LIN {X 43.957,Y 37.252,Z 55.996,A 180.000,B 0.000,C 180.000} C_DIS
LIN {X 43.920,Y 37.565,Z 55.994,A 180.000,B 0.000,C 180.000} C_DIS
LIN {X 43.871,Y 37.876,Z 55.991,A 180.000,B 0.000,C 180.000} C_DIS
LIN {X 43.804,Y 38.184,Z 55.988,A 180.000,B 0.000,C 180.000} C_DIS
LIN {X 43.727,Y 38.489,Z 55.985,A 180.000,B 0.000,C 180.000} C_DIS
LIN {X 43.639,Y 38.792,Z 55.981,A 180.000,B 0.000,C 180.000} C_DIS
LIN {X 43.534,Y 39.089,Z 55.977,A 180.000,B 0.000,C 180.000} C_DIS
LIN {X 43.420,Y 39.382,Z 55.972,A 180.000,B 0.000,C 180.000} C_DIS
LIN {X 43.357,Y 39.527,Z 55.969,A 180.000,B 0.000,C 180.000} C_DIS
LIN {X 43.294,Y 39.671,Z 55.967,A 180.000,B 0.000,C 180.000} C_DIS
LIN {X 43.224,Y 39.812,Z 55.964,A 180.000,B 0.000,C 180.000} C_DIS
LIN {X 43.153,Y 39.952,Z 55.961,A 180.000,B 0.000,C 180.000} C_DIS
LIN {X 43.081,Y 40.093,Z 55.959,A 180.000,B 0.000,C 180.000} C_DIS
LIN {X 43.002,Y 40.229,Z 55.956,A 180.000,B 0.000,C 180.000} C_DIS
LIN {X 42.922,Y 40.365,Z 55.952,A 180.000,B 0.000,C 180.000} C_DIS
LIN {X 42.842,Y 40.500,Z 55.949,A 180.000,B 0.000,C 180.000} C_DIS
LIN {X 42.755,Y 40.631,Z 55.946,A 180.000,B 0.000,C 180.000} C_DIS
LIN {X 42.666,Y 40.761,Z 55.943,A 180.000,B 0.000,C 180.000} C_DIS
LIN {X 42.577,Y 40.892,Z 55.939,A 180.000,B 0.000,C 180.000} C_DIS
LIN {X 42.482,Y 41.017,Z 55.936,A 180.000,B 0.000,C 180.000} C_DIS
LIN {X 42.385,Y 41.141,Z 55.932,A 180.000,B 0.000,C 180.000} C_DIS
LIN {X 42.289,Y 41.266,Z 55.928,A 180.000,B 0.000,C 180.000} C_DIS
LIN {X 42.185,Y 41.385,Z 55.925,A 180.000,B 0.000,C 180.000} C_DIS
LIN {X 42.081,Y 41.503,Z 55.921,A 180.000,B 0.000,C 180.000} C_DIS
LIN {X 41.977,Y 41.621,Z 55.917,A 180.000,B 0.000,C 180.000} C_DIS
LIN {X 41.867,Y 41.733,Z 55.913,A 180.000,B 0.000,C 180.000} C_DIS
LIN {X 41.755,Y 41.844,Z 55.909,A 180.000,B 0.000,C 180.000} C_DIS
LIN {X 41.644,Y 41.956,Z 55.905,A 180.000,B 0.000,C 180.000} C_DIS
LIN {X 41.526,Y 42.061,Z 55.900,A 180.000,B 0.000,C 180.000} C_DIS
LIN {X 41.408,Y 42.165,Z 55.896,A 180.000,B 0.000,C 180.000} C_DIS
LIN {X 41.290,Y 42.269,Z 55.892,A 180.000,B 0.000,C 180.000} C_DIS
LIN {X 41.166,Y 42.366,Z 55.887,A 180.000,B 0.000,C 180.000} C_DIS
LIN {X 41.042,Y 42.463,Z 55.883,A 180.000,B 0.000,C 180.000} C_DIS
LIN {X 40.917,Y 42.559,Z 55.878,A 180.000,B 0.000,C 180.000} C_DIS
LIN {X 40.787,Y 42.648,Z 55.873,A 180.000,B 0.000,C 180.000} C_DIS
LIN {X 40.657,Y 42.737,Z 55.869,A 180.000,B 0.000,C 180.000} C_DIS
LIN {X 40.527,Y 42.826,Z 55.864,A 180.000,B 0.000,C 180.000} C_DIS
LIN {X 40.391,Y 42.906,Z 55.859,A 180.000,B 0.000,C 180.000} C_DIS
LIN {X 40.256,Y 42.986,Z 55.854,A 180.000,B 0.000,C 180.000} C_DIS
LIN {X 40.188,Y 43.027,Z 55.851,A 180.000,B 0.000,C 180.000} C_DIS
LIN {X 40.120,Y 43.067,Z 55.849,A 180.000,B 0.000,C 180.000} C_DIS
LIN {X 40.050,Y 43.103,Z 55.846,A 180.000,B 0.000,C 180.000} C_DIS
LIN {X 39.980,Y 43.139,Z 55.844,A 180.000,B 0.000,C 180.000} C_DIS
LIN {X 39.910,Y 43.174,Z 55.841,A 180.000,B 0.000,C 180.000} C_DIS
LIN {X 39.840,Y 43.210,Z 55.839,A 180.000,B 0.000,C 180.000} C_DIS
LIN {X 39.770,Y 43.246,Z 55.836,A 180.000,B 0.000,C 180.000} C_DIS
LIN {X 39.700,Y 43.282,Z 55.833,A 180.000,B 0.000,C 180.000} C_DIS
LIN {X 39.627,Y 43.313,Z 55.831,A 180.000,B 0.000,C 180.000} C_DIS
LIN {X 39.483,Y 43.376,Z 55.825,A 180.000,B 0.000,C 180.000} C_DIS
LIN {X 39.338,Y 43.438,Z 55.820,A 180.000,B 0.000,C 180.000} C_DIS
LIN {X 39.266,Y 43.470,Z 55.817,A 180.000,B 0.000,C 180.000} C_DIS
LIN {X 39.192,Y 43.497,Z 55.815,A 180.000,B 0.000,C 180.000} C_DIS
LIN {X 39.044,Y 43.550,Z 55.809,A 180.000,B 0.000,C 180.000} C_DIS
LIN {X 38.970,Y 43.577,Z 55.806,A 180.000,B 0.000,C 180.000} C_DIS
LIN {X 38.822,Y 43.630,Z 55.801,A 180.000,B 0.000,C 180.000} C_DIS
LIN {X 38.746,Y 43.652,Z 55.798,A 180.000,B 0.000,C 180.000} C_DIS
LIN {X 38.670,Y 43.674,Z 55.796,A 180.000,B 0.000,C 180.000} C_DIS
LIN {X 38.519,Y 43.718,Z 55.790,A 180.000,B 0.000,C 180.000} C_DIS
LIN {X 38.368,Y 43.762,Z 55.785,A 180.000,B 0.000,C 180.000} C_DIS
LIN {X 38.291,Y 43.780,Z 55.782,A 180.000,B 0.000,C 180.000} C_DIS
LIN {X 38.137,Y 43.814,Z 55.776,A 180.000,B 0.000,C 180.000} C_DIS
LIN {X 38.060,Y 43.831,Z 55.774,A 180.000,B 0.000,C 180.000} C_DIS
LIN {X 37.907,Y 43.866,Z 55.768,A 180.000,B 0.000,C 180.000} C_DIS
LIN {X 37.829,Y 43.878,Z 55.765,A 180.000,B 0.000,C 180.000} C_DIS
LIN {X 37.751,Y 43.890,Z 55.763,A 180.000,B 0.000,C 180.000} C_DIS
LIN {X 37.596,Y 43.915,Z 55.757,A 180.000,B 0.000,C 180.000} C_DIS
LIN {X 37.440,Y 43.940,Z 55.752,A 180.000,B 0.000,C 180.000} C_DIS
LIN {X 37.362,Y 43.947,Z 55.749,A 180.000,B 0.000,C 180.000} C_DIS
LIN {X 37.205,Y 43.962,Z 55.743,A 180.000,B 0.000,C 180.000} C_DIS
LIN {X 37.126,Y 43.969,Z 55.741,A 180.000,B 0.000,C 180.000} C_DIS
LIN {X 37.048,Y 43.977,Z 55.738,A 180.000,B 0.000,C 180.000} C_DIS
LIN {X 36.970,Y 43.984,Z 55.735,A 180.000,B 0.000,C 180.000} C_DIS
LIN {X 36.576,Y 43.996,Z 55.721,A 180.000,B 0.000,C 180.000} C_DIS
LIN {X 36.497,Y 43.999,Z 55.719,A 180.000,B 0.000,C 180.000} C_DIS
LIN {X 36.340,Y 43.994,Z 55.713,A 180.000,B 0.000,C 180.000} C_DIS
LIN {X 36.104,Y 43.986,Z 55.705,A 180.000,B 0.000,C 180.000} C_DIS
LIN {X 36.025,Y 43.984,Z 55.702,A 180.000,B 0.000,C 180.000} C_DIS
LIN {X 35.633,Y 43.947,Z 55.688,A 180.000,B 0.000,C 180.000} C_DIS
LIN {X 35.555,Y 43.939,Z 55.686,A 180.000,B 0.000,C 180.000} C_DIS
LIN {X 35.399,Y 43.914,Z 55.680,A 180.000,B 0.000,C 180.000} C_DIS
LIN {X 35.166,Y 43.877,Z 55.672,A 180.000,B 0.000,C 180.000} C_DIS
LIN {X 35.088,Y 43.864,Z 55.669,A 180.000,B 0.000,C 180.000} C_DIS
LIN {X 34.704,Y 43.778,Z 55.655,A 180.000,B 0.000,C 180.000} C_DIS
LIN {X 34.627,Y 43.761,Z 55.653,A 180.000,B 0.000,C 180.000} C_DIS
LIN {X 34.400,Y 43.695,Z 55.644,A 180.000,B 0.000,C 180.000} C_DIS
LIN {X 34.249,Y 43.651,Z 55.639,A 180.000,B 0.000,C 180.000} C_DIS
LIN {X 34.173,Y 43.628,Z 55.636,A 180.000,B 0.000,C 180.000} C_DIS
LIN {X 33.803,Y 43.495,Z 55.622,A 180.000,B 0.000,C 180.000} C_DIS
LIN {X 33.729,Y 43.468,Z 55.620,A 180.000,B 0.000,C 180.000} C_DIS
LIN {X 33.512,Y 43.374,Z 55.611,A 180.000,B 0.000,C 180.000} C_DIS
LIN {X 33.368,Y 43.311,Z 55.606,A 180.000,B 0.000,C 180.000} C_DIS
LIN {X 33.296,Y 43.279,Z 55.603,A 180.000,B 0.000,C 180.000} C_DIS
LIN {X 32.945,Y 43.100,Z 55.589,A 180.000,B 0.000,C 180.000} C_DIS
LIN {X 32.875,Y 43.064,Z 55.587,A 180.000,B 0.000,C 180.000} C_DIS
LIN {X 32.536,Y 42.863,Z 55.573,A 180.000,B 0.000,C 180.000} C_DIS
LIN {X 32.469,Y 42.822,Z 55.570,A 180.000,B 0.000,C 180.000} C_DIS
LIN {X 32.143,Y 42.601,Z 55.556,A 180.000,B 0.000,C 180.000} C_DIS
LIN {X 32.079,Y 42.556,Z 55.554,A 180.000,B 0.000,C 180.000} C_DIS
LIN {X 31.767,Y 42.315,Z 55.540,A 180.000,B 0.000,C 180.000} C_DIS
LIN {X 31.706,Y 42.265,Z 55.537,A 180.000,B 0.000,C 180.000} C_DIS
LIN {X 31.410,Y 42.005,Z 55.523,A 180.000,B 0.000,C 180.000} C_DIS
LIN {X 31.352,Y 41.952,Z 55.521,A 180.000,B 0.000,C 180.000} C_DIS
LIN {X 31.074,Y 41.673,Z 55.507,A 180.000,B 0.000,C 180.000} C_DIS
LIN {X 31.019,Y 41.617,Z 55.504,A 180.000,B 0.000,C 180.000} C_DIS
LIN {X 30.759,Y 41.321,Z 55.490,A 180.000,B 0.000,C 180.000} C_DIS
LIN {X 30.708,Y 41.261,Z 55.488,A 180.000,B 0.000,C 180.000} C_DIS
LIN {X 30.466,Y 40.950,Z 55.474,A 180.000,B 0.000,C 180.000} C_DIS
LIN {X 30.419,Y 40.887,Z 55.471,A 180.000,B 0.000,C 180.000} C_DIS
LIN {X 30.198,Y 40.561,Z 55.457,A 180.000,B 0.000,C 180.000} C_DIS
LIN {X 30.155,Y 40.495,Z 55.455,A 180.000,B 0.000,C 180.000} C_DIS
LIN {X 29.955,Y 40.156,Z 55.441,A 180.000,B 0.000,C 180.000} C_DIS
LIN {X 29.916,Y 40.088,Z 55.438,A 180.000,B 0.000,C 180.000} C_DIS
LIN {X 29.737,Y 39.737,Z 55.424,A 180.000,B 0.000,C 180.000} C_DIS
LIN {X 29.703,Y 39.666,Z 55.422,A 180.000,B 0.000,C 180.000} C_DIS
LIN {X 29.547,Y 39.305,Z 55.408,A 180.000,B 0.000,C 180.000} C_DIS
LIN {X 29.517,Y 39.232,Z 55.405,A 180.000,B 0.000,C 180.000} C_DIS
LIN {X 29.384,Y 38.861,Z 55.391,A 180.000,B 0.000,C 180.000} C_DIS
LIN {X 29.359,Y 38.786,Z 55.389,A 180.000,B 0.000,C 180.000} C_DIS
LIN {X 29.293,Y 38.559,Z 55.380,A 180.000,B 0.000,C 180.000} C_DIS
LIN {X 29.249,Y 38.408,Z 55.375,A 180.000,B 0.000,C 180.000} C_DIS
LIN {X 29.229,Y 38.332,Z 55.372,A 180.000,B 0.000,C 180.000} C_DIS
LIN {X 29.144,Y 37.948,Z 55.358,A 180.000,B 0.000,C 180.000} C_DIS
LIN {X 29.129,Y 37.870,Z 55.356,A 180.000,B 0.000,C 180.000} C_DIS
LIN {X 29.092,Y 37.637,Z 55.347,A 180.000,B 0.000,C 180.000} C_DIS
LIN {X 29.067,Y 37.481,Z 55.342,A 180.000,B 0.000,C 180.000} C_DIS
LIN {X 29.057,Y 37.403,Z 55.339,A 180.000,B 0.000,C 180.000} C_DIS
LIN {X 29.020,Y 37.011,Z 55.325,A 180.000,B 0.000,C 180.000} C_DIS
LIN {X 29.015,Y 36.933,Z 55.323,A 180.000,B 0.000,C 180.000} C_DIS
LIN {X 29.010,Y 36.775,Z 55.317,A 180.000,B 0.000,C 180.000} C_DIS
LIN {X 29.002,Y 36.539,Z 55.309,A 180.000,B 0.000,C 180.000} C_DIS
LIN {X 29.002,Y 36.460,Z 55.306,A 180.000,B 0.000,C 180.000} C_DIS
LIN {X 29.015,Y 36.067,Z 55.292,A 180.000,B 0.000,C 180.000} C_DIS
LIN {X 29.020,Y 35.988,Z 55.290,A 180.000,B 0.000,C 180.000} C_DIS
LIN {X 29.035,Y 35.831,Z 55.284,A 180.000,B 0.000,C 180.000} C_DIS
LIN {X 29.057,Y 35.596,Z 55.276,A 180.000,B 0.000,C 180.000} C_DIS
LIN {X 29.067,Y 35.518,Z 55.273,A 180.000,B 0.000,C 180.000} C_DIS
LIN {X 29.104,Y 35.285,Z 55.265,A 180.000,B 0.000,C 180.000} C_DIS
LIN {X 29.129,Y 35.129,Z 55.259,A 180.000,B 0.000,C 180.000} C_DIS
LIN {X 29.144,Y 35.052,Z 55.257,A 180.000,B 0.000,C 180.000} C_DIS
LIN {X 29.178,Y 34.898,Z 55.251,A 180.000,B 0.000,C 180.000} C_DIS
LIN {X 29.230,Y 34.668,Z 55.243,A 180.000,B 0.000,C 180.000} C_DIS
LIN {X 29.250,Y 34.591,Z 55.240,A 180.000,B 0.000,C 180.000} C_DIS
LIN {X 29.315,Y 34.365,Z 55.232,A 180.000,B 0.000,C 180.000} C_DIS
LIN {X 29.359,Y 34.213,Z 55.226,A 180.000,B 0.000,C 180.000} C_DIS
LIN {X 29.384,Y 34.139,Z 55.224,A 180.000,B 0.000,C 180.000} C_DIS
LIN {X 29.438,Y 33.990,Z 55.218,A 180.000,B 0.000,C 180.000} C_DIS
LIN {X 29.518,Y 33.768,Z 55.210,A 180.000,B 0.000,C 180.000} C_DIS
LIN {X 29.547,Y 33.695,Z 55.207,A 180.000,B 0.000,C 180.000} C_DIS
LIN {X 29.641,Y 33.478,Z 55.199,A 180.000,B 0.000,C 180.000} C_DIS
LIN {X 29.703,Y 33.334,Z 55.193,A 180.000,B 0.000,C 180.000} C_DIS
LIN {X 29.738,Y 33.263,Z 55.191,A 180.000,B 0.000,C 180.000} C_DIS
LIN {X 29.809,Y 33.122,Z 55.185,A 180.000,B 0.000,C 180.000} C_DIS
LIN {X 29.881,Y 32.982,Z 55.180,A 180.000,B 0.000,C 180.000} C_DIS
LIN {X 29.916,Y 32.912,Z 55.177,A 180.000,B 0.000,C 180.000} C_DIS
LIN {X 29.955,Y 32.843,Z 55.174,A 180.000,B 0.000,C 180.000} C_DIS
LIN {X 30.035,Y 32.708,Z 55.169,A 180.000,B 0.000,C 180.000} C_DIS
LIN {X 30.115,Y 32.572,Z 55.164,A 180.000,B 0.000,C 180.000} C_DIS
LIN {X 30.155,Y 32.504,Z 55.161,A 180.000,B 0.000,C 180.000} C_DIS
LIN {X 30.198,Y 32.438,Z 55.159,A 180.000,B 0.000,C 180.000} C_DIS
LIN {X 30.243,Y 32.373,Z 55.156,A 180.000,B 0.000,C 180.000} C_DIS
LIN {X 30.287,Y 32.308,Z 55.154,A 180.000,B 0.000,C 180.000} C_DIS
LIN {X 30.331,Y 32.243,Z 55.151,A 180.000,B 0.000,C 180.000} C_DIS
LIN {X 30.375,Y 32.178,Z 55.149,A 180.000,B 0.000,C 180.000} C_DIS
LIN {X 30.467,Y 32.049,Z 55.144,A 180.000,B 0.000,C 180.000} C_DIS
LIN {X 30.563,Y 31.925,Z 55.139,A 180.000,B 0.000,C 180.000} C_DIS
LIN {X 30.660,Y 31.800,Z 55.134,A 180.000,B 0.000,C 180.000} C_DIS
LIN {X 30.759,Y 31.678,Z 55.129,A 180.000,B 0.000,C 180.000} C_DIS
LIN {X 30.863,Y 31.560,Z 55.124,A 180.000,B 0.000,C 180.000} C_DIS
LIN {X 30.967,Y 31.442,Z 55.120,A 180.000,B 0.000,C 180.000} C_DIS
LIN {X 31.074,Y 31.326,Z 55.115,A 180.000,B 0.000,C 180.000} C_DIS
LIN {X 31.186,Y 31.215,Z 55.111,A 180.000,B 0.000,C 180.000} C_DIS
LIN {X 31.297,Y 31.103,Z 55.106,A 180.000,B 0.000,C 180.000} C_DIS
LIN {X 31.411,Y 30.995,Z 55.102,A 180.000,B 0.000,C 180.000} C_DIS
LIN {X 31.529,Y 30.891,Z 55.097,A 180.000,B 0.000,C 180.000} C_DIS
LIN {X 31.647,Y 30.786,Z 55.093,A 180.000,B 0.000,C 180.000} C_DIS
LIN {X 31.768,Y 30.685,Z 55.089,A 180.000,B 0.000,C 180.000} C_DIS
LIN {X 31.892,Y 30.589,Z 55.085,A 180.000,B 0.000,C 180.000} C_DIS
LIN {X 32.017,Y 30.492,Z 55.081,A 180.000,B 0.000,C 180.000} C_DIS
LIN {X 32.144,Y 30.399,Z 55.077,A 180.000,B 0.000,C 180.000} C_DIS
LIN {X 32.274,Y 30.310,Z 55.073,A 180.000,B 0.000,C 180.000} C_DIS
LIN {X 32.404,Y 30.222,Z 55.070,A 180.000,B 0.000,C 180.000} C_DIS
LIN {X 32.537,Y 30.136,Z 55.066,A 180.000,B 0.000,C 180.000} C_DIS
LIN {X 32.672,Y 30.056,Z 55.062,A 180.000,B 0.000,C 180.000} C_DIS
LIN {X 32.808,Y 29.976,Z 55.059,A 180.000,B 0.000,C 180.000} C_DIS
LIN {X 32.945,Y 29.899,Z 55.056,A 180.000,B 0.000,C 180.000} C_DIS
LIN {X 33.086,Y 29.828,Z 55.052,A 180.000,B 0.000,C 180.000} C_DIS
LIN {X 33.226,Y 29.756,Z 55.049,A 180.000,B 0.000,C 180.000} C_DIS
LIN {X 33.368,Y 29.689,Z 55.046,A 180.000,B 0.000,C 180.000} C_DIS
LIN {X 33.513,Y 29.626,Z 55.043,A 180.000,B 0.000,C 180.000} C_DIS
LIN {X 33.657,Y 29.563,Z 55.040,A 180.000,B 0.000,C 180.000} C_DIS
LIN {X 33.803,Y 29.505,Z 55.037,A 180.000,B 0.000,C 180.000} C_DIS
LIN {X 33.952,Y 29.451,Z 55.034,A 180.000,B 0.000,C 180.000} C_DIS
LIN {X 34.100,Y 29.398,Z 55.032,A 180.000,B 0.000,C 180.000} C_DIS
LIN {X 34.249,Y 29.349,Z 55.029,A 180.000,B 0.000,C 180.000} C_DIS
LIN {X 34.401,Y 29.305,Z 55.027,A 180.000,B 0.000,C 180.000} C_DIS
LIN {X 34.704,Y 29.221,Z 55.022,A 180.000,B 0.000,C 180.000} C_DIS
LIN {X 35.012,Y 29.153,Z 55.018,A 180.000,B 0.000,C 180.000} C_DIS
LIN {X 35.322,Y 29.098,Z 55.014,A 180.000,B 0.000,C 180.000} C_DIS
LIN {X 35.634,Y 29.053,Z 55.011,A 180.000,B 0.000,C 180.000} C_DIS
LIN {X 35.947,Y 29.024,Z 55.008,A 180.000,B 0.000,C 180.000} C_DIS
LIN {X 36.262,Y 29.009,Z 55.005,A 180.000,B 0.000,C 180.000} C_DIS
LIN {X 36.577,Y 29.004,Z 55.003,A 180.000,B 0.000,C 180.000} C_DIS
LIN {X 36.891,Y 29.014,Z 55.002,A 180.000,B 0.000,C 180.000} C_DIS
LIN {X 37.205,Y 29.038,Z 55.001,A 180.000,B 0.000,C 180.000} C_DIS
LIN {X 37.518,Y 29.073,Z 55.000,A 180.000,B 0.000,C 180.000} C_DIS
LIN {X 37.748,Y 29.109,Z 55.000,A 180.000,B 0.000,C 180.000} C_DIS
; Cutting Move Starts
LIN {X 37.902,Y 29.134,Z 55.000,A 180.000,B 0.000,C 180.000} C_DIS
LIN {X 37.944,Y 29.143,Z 55.000,A 180.000,B 0.000,C 180.000} C_DIS
LIN {X 38.260,Y 29.213,Z 55.000,A 180.000,B 0.000,C 180.000} C_DIS
LIN {X 38.439,Y 29.258,Z 55.000,A 180.000,B 0.000,C 180.000} C_DIS
LIN {X 38.796,Y 29.362,Z 55.000,A 180.000,B 0.000,C 180.000} C_DIS
LIN {X 38.975,Y 29.425,Z 55.000,A 180.000,B 0.000,C 180.000} C_DIS
LIN {X 39.184,Y 29.500,Z 55.000,A 180.000,B 0.000,C 180.000} C_DIS
LIN {X 39.333,Y 29.559,Z 55.000,A 180.000,B 0.000,C 180.000} C_DIS
LIN {X 39.690,Y 29.714,Z 55.000,A 180.000,B 0.000,C 180.000} C_DIS
LIN {X 39.869,Y 29.805,Z 55.000,A 180.000,B 0.000,C 180.000} C_DIS
LIN {X 40.048,Y 29.896,Z 55.000,A 180.000,B 0.000,C 180.000} C_DIS
LIN {X 40.226,Y 29.996,Z 55.000,A 180.000,B 0.000,C 180.000} C_DIS
LIN {X 40.405,Y 30.102,Z 55.000,A 180.000,B 0.000,C 180.000} C_DIS
LIN {X 40.584,Y 30.213,Z 55.000,A 180.000,B 0.000,C 180.000} C_DIS
LIN {X 40.850,Y 30.394,Z 55.000,A 180.000,B 0.000,C 180.000} C_DIS
LIN {X 40.942,Y 30.460,Z 55.000,A 180.000,B 0.000,C 180.000} C_DIS
LIN {X 41.120,Y 30.598,Z 55.000,A 180.000,B 0.000,C 180.000} C_DIS
LIN {X 41.299,Y 30.739,Z 55.000,A 180.000,B 0.000,C 180.000} C_DIS
LIN {X 41.516,Y 30.930,Z 55.000,A 180.000,B 0.000,C 180.000} C_DIS
LIN {X 41.657,Y 31.057,Z 55.000,A 180.000,B 0.000,C 180.000} C_DIS
LIN {X 41.888,Y 31.288,Z 55.000,A 180.000,B 0.000,C 180.000} C_DIS
LIN {X 42.014,Y 31.421,Z 55.000,A 180.000,B 0.000,C 180.000} C_DIS
LIN {X 42.212,Y 31.646,Z 55.000,A 180.000,B 0.000,C 180.000} C_DIS
LIN {X 42.359,Y 31.824,Z 55.000,A 180.000,B 0.000,C 180.000} C_DIS
LIN {X 42.550,Y 32.072,Z 55.000,A 180.000,B 0.000,C 180.000} C_DIS
LIN {X 42.627,Y 32.182,Z 55.000,A 180.000,B 0.000,C 180.000} C_DIS
LIN {X 42.749,Y 32.361,Z 55.000,A 180.000,B 0.000,C 180.000} C_DIS
LIN {X 42.865,Y 32.539,Z 55.000,A 180.000,B 0.000,C 180.000} C_DIS
LIN {X 42.971,Y 32.718,Z 55.000,A 180.000,B 0.000,C 180.000} C_DIS
LIN {X 43.076,Y 32.897,Z 55.000,A 180.000,B 0.000,C 180.000} C_DIS
LIN {X 43.266,Y 33.269,Z 55.000,A 180.000,B 0.000,C 180.000} C_DIS
LIN {X 43.340,Y 33.433,Z 55.000,A 180.000,B 0.000,C 180.000} C_DIS
LIN {X 43.444,Y 33.675,Z 55.000,A 180.000,B 0.000,C 180.000} C_DIS
LIN {X 43.491,Y 33.791,Z 55.000,A 180.000,B 0.000,C 180.000} C_DIS
LIN {X 43.623,Y 34.159,Z 55.000,A 180.000,B 0.000,C 180.000} C_DIS
LIN {X 43.674,Y 34.327,Z 55.000,A 180.000,B 0.000,C 180.000} C_DIS
LIN {X 43.726,Y 34.506,Z 55.000,A 180.000,B 0.000,C 180.000} C_DIS
LIN {X 43.774,Y 34.685,Z 55.000,A 180.000,B 0.000,C 180.000} C_DIS
LIN {X 43.854,Y 35.042,Z 55.000,A 180.000,B 0.000,C 180.000} C_DIS
LIN {X 43.886,Y 35.221,Z 55.000,A 180.000,B 0.000,C 180.000} C_DIS
LIN {X 43.914,Y 35.400,Z 55.000,A 180.000,B 0.000,C 180.000} C_DIS
LIN {X 43.941,Y 35.578,Z 55.000,A 180.000,B 0.000,C 180.000} C_DIS
LIN {X 43.981,Y 35.994,Z 55.000,A 180.000,B 0.000,C 180.000} C_DIS
LIN {X 43.987,Y 36.115,Z 55.000,A 180.000,B 0.000,C 180.000} C_DIS
LIN {X 43.998,Y 36.472,Z 55.000,A 180.000,B 0.000,C 180.000} C_DIS
LIN {X 43.994,Y 36.651,Z 55.000,A 180.000,B 0.000,C 180.000} C_DIS
LIN {X 43.988,Y 36.830,Z 55.000,A 180.000,B 0.000,C 180.000} C_DIS
LIN {X 43.981,Y 37.006,Z 55.000,A 180.000,B 0.000,C 180.000} C_DIS
LIN {X 43.947,Y 37.366,Z 55.000,A 180.000,B 0.000,C 180.000} C_DIS
LIN {X 43.923,Y 37.545,Z 55.000,A 180.000,B 0.000,C 180.000} C_DIS
LIN {X 43.866,Y 37.902,Z 55.000,A 180.000,B 0.000,C 180.000} C_DIS
LIN {X 43.827,Y 38.081,Z 55.000,A 180.000,B 0.000,C 180.000} C_DIS
LIN {X 43.787,Y 38.260,Z 55.000,A 180.000,B 0.000,C 180.000} C_DIS
LIN {X 43.742,Y 38.439,Z 55.000,A 180.000,B 0.000,C 180.000} C_DIS
LIN {X 43.638,Y 38.796,Z 55.000,A 180.000,B 0.000,C 180.000} C_DIS
LIN {X 43.623,Y 38.841,Z 55.000,A 180.000,B 0.000,C 180.000} C_DIS
LIN {X 43.511,Y 39.154,Z 55.000,A 180.000,B 0.000,C 180.000} C_DIS
LIN {X 43.444,Y 39.325,Z 55.000,A 180.000,B 0.000,C 180.000} C_DIS
LIN {X 43.286,Y 39.690,Z 55.000,A 180.000,B 0.000,C 180.000} C_DIS
LIN {X 43.266,Y 39.731,Z 55.000,A 180.000,B 0.000,C 180.000} C_DIS
LIN {X 43.087,Y 40.082,Z 55.000,A 180.000,B 0.000,C 180.000} C_DIS
LIN {X 43.004,Y 40.226,Z 55.000,A 180.000,B 0.000,C 180.000} C_DIS
LIN {X 42.898,Y 40.405,Z 55.000,A 180.000,B 0.000,C 180.000} C_DIS
LIN {X 42.787,Y 40.584,Z 55.000,A 180.000,B 0.000,C 180.000} C_DIS
LIN {X 42.665,Y 40.763,Z 55.000,A 180.000,B 0.000,C 180.000} C_DIS
LIN {X 42.550,Y 40.928,Z 55.000,A 180.000,B 0.000,C 180.000} C_DIS
LIN {X 42.372,Y 41.159,Z 55.000,A 180.000,B 0.000,C 180.000} C_DIS
LIN {X 42.261,Y 41.299,Z 55.000,A 180.000,B 0.000,C 180.000} C_DIS
LIN {X 42.014,Y 41.579,Z 55.000,A 180.000,B 0.000,C 180.000} C_DIS
LIN {X 41.943,Y 41.657,Z 55.000,A 180.000,B 0.000,C 180.000} C_DIS
LIN {X 41.657,Y 41.943,Z 55.000,A 180.000,B 0.000,C 180.000} C_DIS
LIN {X 41.579,Y 42.014,Z 55.000,A 180.000,B 0.000,C 180.000} C_DIS
LIN {X 41.299,Y 42.261,Z 55.000,A 180.000,B 0.000,C 180.000} C_DIS
LIN {X 41.159,Y 42.372,Z 55.000,A 180.000,B 0.000,C 180.000} C_DIS
LIN {X 40.928,Y 42.550,Z 55.000,A 180.000,B 0.000,C 180.000} C_DIS
LIN {X 40.763,Y 42.665,Z 55.000,A 180.000,B 0.000,C 180.000} C_DIS
LIN {X 40.584,Y 42.787,Z 55.000,A 180.000,B 0.000,C 180.000} C_DIS
LIN {X 40.405,Y 42.898,Z 55.000,A 180.000,B 0.000,C 180.000} C_DIS
LIN {X 40.226,Y 43.004,Z 55.000,A 180.000,B 0.000,C 180.000} C_DIS
LIN {X 40.082,Y 43.087,Z 55.000,A 180.000,B 0.000,C 180.000} C_DIS
LIN {X 39.731,Y 43.266,Z 55.000,A 180.000,B 0.000,C 180.000} C_DIS
LIN {X 39.690,Y 43.286,Z 55.000,A 180.000,B 0.000,C 180.000} C_DIS
LIN {X 39.325,Y 43.444,Z 55.000,A 180.000,B 0.000,C 180.000} C_DIS
LIN {X 39.154,Y 43.511,Z 55.000,A 180.000,B 0.000,C 180.000} C_DIS
LIN {X 38.841,Y 43.623,Z 55.000,A 180.000,B 0.000,C 180.000} C_DIS
LIN {X 38.796,Y 43.638,Z 55.000,A 180.000,B 0.000,C 180.000} C_DIS
LIN {X 38.439,Y 43.742,Z 55.000,A 180.000,B 0.000,C 180.000} C_DIS
LIN {X 38.260,Y 43.787,Z 55.000,A 180.000,B 0.000,C 180.000} C_DIS
LIN {X 38.081,Y 43.827,Z 55.000,A 180.000,B 0.000,C 180.000} C_DIS
LIN {X 37.902,Y 43.866,Z 55.000,A 180.000,B 0.000,C 180.000} C_DIS
LIN {X 37.545,Y 43.923,Z 55.000,A 180.000,B 0.000,C 180.000} C_DIS
LIN {X 37.366,Y 43.947,Z 55.000,A 180.000,B 0.000,C 180.000} C_DIS
LIN {X 37.006,Y 43.981,Z 55.000,A 180.000,B 0.000,C 180.000} C_DIS
LIN {X 36.830,Y 43.988,Z 55.000,A 180.000,B 0.000,C 180.000} C_DIS
LIN {X 36.651,Y 43.994,Z 55.000,A 180.000,B 0.000,C 180.000} C_DIS
LIN {X 36.472,Y 43.998,Z 55.000,A 180.000,B 0.000,C 180.000} C_DIS
LIN {X 36.115,Y 43.987,Z 55.000,A 180.000,B 0.000,C 180.000} C_DIS
LIN {X 35.994,Y 43.981,Z 55.000,A 180.000,B 0.000,C 180.000} C_DIS
LIN {X 35.578,Y 43.941,Z 55.000,A 180.000,B 0.000,C 180.000} C_DIS
LIN {X 35.400,Y 43.914,Z 55.000,A 180.000,B 0.000,C 180.000} C_DIS
LIN {X 35.221,Y 43.886,Z 55.000,A 180.000,B 0.000,C 180.000} C_DIS
LIN {X 35.042,Y 43.854,Z 55.000,A 180.000,B 0.000,C 180.000} C_DIS
LIN {X 34.685,Y 43.774,Z 55.000,A 180.000,B 0.000,C 180.000} C_DIS
LIN {X 34.506,Y 43.726,Z 55.000,A 180.000,B 0.000,C 180.000} C_DIS
LIN {X 34.327,Y 43.674,Z 55.000,A 180.000,B 0.000,C 180.000} C_DIS
LIN {X 34.159,Y 43.623,Z 55.000,A 180.000,B 0.000,C 180.000} C_DIS
LIN {X 33.791,Y 43.491,Z 55.000,A 180.000,B 0.000,C 180.000} C_DIS
LIN {X 33.675,Y 43.444,Z 55.000,A 180.000,B 0.000,C 180.000} C_DIS
LIN {X 33.433,Y 43.340,Z 55.000,A 180.000,B 0.000,C 180.000} C_DIS
LIN {X 33.269,Y 43.266,Z 55.000,A 180.000,B 0.000,C 180.000} C_DIS
LIN {X 32.897,Y 43.076,Z 55.000,A 180.000,B 0.000,C 180.000} C_DIS
LIN {X 32.718,Y 42.971,Z 55.000,A 180.000,B 0.000,C 180.000} C_DIS
LIN {X 32.539,Y 42.865,Z 55.000,A 180.000,B 0.000,C 180.000} C_DIS
LIN {X 32.361,Y 42.749,Z 55.000,A 180.000,B 0.000,C 180.000} C_DIS
LIN {X 32.182,Y 42.627,Z 55.000,A 180.000,B 0.000,C 180.000} C_DIS
LIN {X 32.072,Y 42.550,Z 55.000,A 180.000,B 0.000,C 180.000} C_DIS
LIN {X 31.824,Y 42.359,Z 55.000,A 180.000,B 0.000,C 180.000} C_DIS
LIN {X 31.646,Y 42.212,Z 55.000,A 180.000,B 0.000,C 180.000} C_DIS
LIN {X 31.421,Y 42.014,Z 55.000,A 180.000,B 0.000,C 180.000} C_DIS
LIN {X 31.288,Y 41.888,Z 55.000,A 180.000,B 0.000,C 180.000} C_DIS
LIN {X 31.057,Y 41.657,Z 55.000,A 180.000,B 0.000,C 180.000} C_DIS
LIN {X 30.930,Y 41.516,Z 55.000,A 180.000,B 0.000,C 180.000} C_DIS
LIN {X 30.739,Y 41.299,Z 55.000,A 180.000,B 0.000,C 180.000} C_DIS
LIN {X 30.598,Y 41.120,Z 55.000,A 180.000,B 0.000,C 180.000} C_DIS
LIN {X 30.460,Y 40.942,Z 55.000,A 180.000,B 0.000,C 180.000} C_DIS
LIN {X 30.394,Y 40.850,Z 55.000,A 180.000,B 0.000,C 180.000} C_DIS
LIN {X 30.213,Y 40.584,Z 55.000,A 180.000,B 0.000,C 180.000} C_DIS
LIN {X 30.102,Y 40.405,Z 55.000,A 180.000,B 0.000,C 180.000} C_DIS
LIN {X 29.996,Y 40.226,Z 55.000,A 180.000,B 0.000,C 180.000} C_DIS
LIN {X 29.896,Y 40.048,Z 55.000,A 180.000,B 0.000,C 180.000} C_DIS
LIN {X 29.805,Y 39.869,Z 55.000,A 180.000,B 0.000,C 180.000} C_DIS
LIN {X 29.714,Y 39.690,Z 55.000,A 180.000,B 0.000,C 180.000} C_DIS
LIN {X 29.559,Y 39.333,Z 55.000,A 180.000,B 0.000,C 180.000} C_DIS
LIN {X 29.500,Y 39.184,Z 55.000,A 180.000,B 0.000,C 180.000} C_DIS
LIN {X 29.425,Y 38.975,Z 55.000,A 180.000,B 0.000,C 180.000} C_DIS
LIN {X 29.362,Y 38.796,Z 55.000,A 180.000,B 0.000,C 180.000} C_DIS
LIN {X 29.258,Y 38.439,Z 55.000,A 180.000,B 0.000,C 180.000} C_DIS
LIN {X 29.213,Y 38.260,Z 55.000,A 180.000,B 0.000,C 180.000} C_DIS
LIN {X 29.143,Y 37.944,Z 55.000,A 180.000,B 0.000,C 180.000} C_DIS
LIN {X 29.134,Y 37.902,Z 55.000,A 180.000,B 0.000,C 180.000} C_DIS
LIN {X 29.077,Y 37.545,Z 55.000,A 180.000,B 0.000,C 180.000} C_DIS
LIN {X 29.053,Y 37.366,Z 55.000,A 180.000,B 0.000,C 180.000} C_DIS
LIN {X 29.020,Y 37.009,Z 55.000,A 180.000,B 0.000,C 180.000} C_DIS
LIN {X 29.012,Y 36.830,Z 55.000,A 180.000,B 0.000,C 180.000} C_DIS
LIN {X 29.006,Y 36.651,Z 55.000,A 180.000,B 0.000,C 180.000} C_DIS
LIN {X 29.002,Y 36.472,Z 55.000,A 180.000,B 0.000,C 180.000} C_DIS
LIN {X 29.013,Y 36.115,Z 55.000,A 180.000,B 0.000,C 180.000} C_DIS
LIN {X 29.025,Y 35.936,Z 55.000,A 180.000,B 0.000,C 180.000} C_DIS
LIN {X 29.059,Y 35.578,Z 55.000,A 180.000,B 0.000,C 180.000} C_DIS
LIN {X 29.086,Y 35.400,Z 55.000,A 180.000,B 0.000,C 180.000} C_DIS
LIN {X 29.114,Y 35.221,Z 55.000,A 180.000,B 0.000,C 180.000} C_DIS
LIN {X 29.143,Y 35.056,Z 55.000,A 180.000,B 0.000,C 180.000} C_DIS
LIN {X 29.226,Y 34.685,Z 55.000,A 180.000,B 0.000,C 180.000} C_DIS
LIN {X 29.274,Y 34.506,Z 55.000,A 180.000,B 0.000,C 180.000} C_DIS
LIN {X 29.326,Y 34.327,Z 55.000,A 180.000,B 0.000,C 180.000} C_DIS
LIN {X 29.381,Y 34.148,Z 55.000,A 180.000,B 0.000,C 180.000} C_DIS
LIN {X 29.509,Y 33.791,Z 55.000,A 180.000,B 0.000,C 180.000} C_DIS
LIN {X 29.583,Y 33.612,Z 55.000,A 180.000,B 0.000,C 180.000} C_DIS
LIN {X 29.679,Y 33.390,Z 55.000,A 180.000,B 0.000,C 180.000} C_DIS
LIN {X 29.742,Y 33.254,Z 55.000,A 180.000,B 0.000,C 180.000} C_DIS
LIN {X 29.924,Y 32.897,Z 55.000,A 180.000,B 0.000,C 180.000} C_DIS
LIN {X 30.029,Y 32.718,Z 55.000,A 180.000,B 0.000,C 180.000} C_DIS
LIN {X 30.135,Y 32.539,Z 55.000,A 180.000,B 0.000,C 180.000} C_DIS
LIN {X 30.215,Y 32.413,Z 55.000,A 180.000,B 0.000,C 180.000} C_DIS
LIN {X 30.394,Y 32.150,Z 55.000,A 180.000,B 0.000,C 180.000} C_DIS
LIN {X 30.503,Y 32.003,Z 55.000,A 180.000,B 0.000,C 180.000} C_DIS
LIN {X 30.641,Y 31.824,Z 55.000,A 180.000,B 0.000,C 180.000} C_DIS
LIN {X 30.752,Y 31.687,Z 55.000,A 180.000,B 0.000,C 180.000} C_DIS
LIN {X 30.945,Y 31.467,Z 55.000,A 180.000,B 0.000,C 180.000} C_DIS
LIN {X 31.109,Y 31.291,Z 55.000,A 180.000,B 0.000,C 180.000} C_DIS
LIN {X 31.291,Y 31.109,Z 55.000,A 180.000,B 0.000,C 180.000} C_DIS
LIN {X 31.467,Y 30.945,Z 55.000,A 180.000,B 0.000,C 180.000} C_DIS
LIN {X 31.687,Y 30.752,Z 55.000,A 180.000,B 0.000,C 180.000} C_DIS
LIN {X 31.824,Y 30.641,Z 55.000,A 180.000,B 0.000,C 180.000} C_DIS
LIN {X 32.003,Y 30.503,Z 55.000,A 180.000,B 0.000,C 180.000} C_DIS
LIN {X 32.150,Y 30.394,Z 55.000,A 180.000,B 0.000,C 180.000} C_DIS
LIN {X 32.413,Y 30.215,Z 55.000,A 180.000,B 0.000,C 180.000} C_DIS
LIN {X 32.539,Y 30.135,Z 55.000,A 180.000,B 0.000,C 180.000} C_DIS
LIN {X 32.718,Y 30.029,Z 55.000,A 180.000,B 0.000,C 180.000} C_DIS
LIN {X 32.897,Y 29.924,Z 55.000,A 180.000,B 0.000,C 180.000} C_DIS
LIN {X 33.254,Y 29.742,Z 55.000,A 180.000,B 0.000,C 180.000} C_DIS
LIN {X 33.390,Y 29.679,Z 55.000,A 180.000,B 0.000,C 180.000} C_DIS
LIN {X 33.612,Y 29.583,Z 55.000,A 180.000,B 0.000,C 180.000} C_DIS
LIN {X 33.791,Y 29.509,Z 55.000,A 180.000,B 0.000,C 180.000} C_DIS
LIN {X 34.148,Y 29.381,Z 55.000,A 180.000,B 0.000,C 180.000} C_DIS
LIN {X 34.327,Y 29.326,Z 55.000,A 180.000,B 0.000,C 180.000} C_DIS
LIN {X 34.506,Y 29.274,Z 55.000,A 180.000,B 0.000,C 180.000} C_DIS
LIN {X 34.685,Y 29.226,Z 55.000,A 180.000,B 0.000,C 180.000} C_DIS
LIN {X 35.056,Y 29.143,Z 55.000,A 180.000,B 0.000,C 180.000} C_DIS
LIN {X 35.221,Y 29.114,Z 55.000,A 180.000,B 0.000,C 180.000} C_DIS
LIN {X 35.400,Y 29.086,Z 55.000,A 180.000,B 0.000,C 180.000} C_DIS
LIN {X 35.578,Y 29.059,Z 55.000,A 180.000,B 0.000,C 180.000} C_DIS
LIN {X 35.936,Y 29.025,Z 55.000,A 180.000,B 0.000,C 180.000} C_DIS
LIN {X 36.115,Y 29.013,Z 55.000,A 180.000,B 0.000,C 180.000} C_DIS
LIN {X 36.472,Y 29.002,Z 55.000,A 180.000,B 0.000,C 180.000} C_DIS
LIN {X 36.651,Y 29.006,Z 55.000,A 180.000,B 0.000,C 180.000} C_DIS
LIN {X 36.830,Y 29.012,Z 55.000,A 180.000,B 0.000,C 180.000} C_DIS
LIN {X 37.009,Y 29.020,Z 55.000,A 180.000,B 0.000,C 180.000} C_DIS
LIN {X 37.366,Y 29.053,Z 55.000,A 180.000,B 0.000,C 180.000} C_DIS
LIN {X 37.545,Y 29.077,Z 55.000,A 180.000,B 0.000,C 180.000} C_DIS
LIN {X 37.748,Y 29.109,Z 55.000,A 180.000,B 0.000,C 180.000} C_DIS
; Link Move Starts
LIN {X 38.057,Y 29.168,Z 55.000,A 180.000,B 0.000,C 180.000} C_DIS
LIN {X 38.365,Y 29.237,Z 54.999,A 180.000,B 0.000,C 180.000} C_DIS
LIN {X 38.667,Y 29.325,Z 54.998,A 180.000,B 0.000,C 180.000} C_DIS
LIN {X 38.967,Y 29.422,Z 54.996,A 180.000,B 0.000,C 180.000} C_DIS
LIN {X 39.263,Y 29.529,Z 54.994,A 180.000,B 0.000,C 180.000} C_DIS
LIN {X 39.552,Y 29.654,Z 54.991,A 180.000,B 0.000,C 180.000} C_DIS
LIN {X 39.837,Y 29.788,Z 54.988,A 180.000,B 0.000,C 180.000} C_DIS
LIN {X 40.117,Y 29.932,Z 54.985,A 180.000,B 0.000,C 180.000} C_DIS
LIN {X 40.389,Y 30.092,Z 54.981,A 180.000,B 0.000,C 180.000} C_DIS
LIN {X 40.654,Y 30.261,Z 54.977,A 180.000,B 0.000,C 180.000} C_DIS
LIN {X 40.915,Y 30.439,Z 54.972,A 180.000,B 0.000,C 180.000} C_DIS
LIN {X 41.039,Y 30.535,Z 54.969,A 180.000,B 0.000,C 180.000} C_DIS
LIN {X 41.163,Y 30.632,Z 54.967,A 180.000,B 0.000,C 180.000} C_DIS
LIN {X 41.288,Y 30.729,Z 54.964,A 180.000,B 0.000,C 180.000} C_DIS
LIN {X 41.406,Y 30.833,Z 54.961,A 180.000,B 0.000,C 180.000} C_DIS
LIN {X 41.524,Y 30.937,Z 54.959,A 180.000,B 0.000,C 180.000} C_DIS
LIN {X 41.641,Y 31.042,Z 54.956,A 180.000,B 0.000,C 180.000} C_DIS
LIN {X 41.753,Y 31.153,Z 54.952,A 180.000,B 0.000,C 180.000} C_DIS
LIN {X 41.864,Y 31.265,Z 54.949,A 180.000,B 0.000,C 180.000} C_DIS
LIN {X 41.975,Y 31.377,Z 54.946,A 180.000,B 0.000,C 180.000} C_DIS
LIN {X 42.079,Y 31.495,Z 54.943,A 180.000,B 0.000,C 180.000} C_DIS
LIN {X 42.183,Y 31.613,Z 54.939,A 180.000,B 0.000,C 180.000} C_DIS
LIN {X 42.287,Y 31.732,Z 54.936,A 180.000,B 0.000,C 180.000} C_DIS
LIN {X 42.383,Y 31.856,Z 54.932,A 180.000,B 0.000,C 180.000} C_DIS
LIN {X 42.480,Y 31.981,Z 54.928,A 180.000,B 0.000,C 180.000} C_DIS
LIN {X 42.576,Y 32.106,Z 54.925,A 180.000,B 0.000,C 180.000} C_DIS
LIN {X 42.664,Y 32.236,Z 54.921,A 180.000,B 0.000,C 180.000} C_DIS
LIN {X 42.753,Y 32.366,Z 54.917,A 180.000,B 0.000,C 180.000} C_DIS
LIN {X 42.840,Y 32.497,Z 54.913,A 180.000,B 0.000,C 180.000} C_DIS
LIN {X 42.921,Y 32.633,Z 54.909,A 180.000,B 0.000,C 180.000} C_DIS
LIN {X 43.001,Y 32.768,Z 54.905,A 180.000,B 0.000,C 180.000} C_DIS
LIN {X 43.080,Y 32.904,Z 54.900,A 180.000,B 0.000,C 180.000} C_DIS
LIN {X 43.151,Y 33.045,Z 54.896,A 180.000,B 0.000,C 180.000} C_DIS
LIN {X 43.223,Y 33.185,Z 54.892,A 180.000,B 0.000,C 180.000} C_DIS
LIN {X 43.293,Y 33.326,Z 54.887,A 180.000,B 0.000,C 180.000} C_DIS
LIN {X 43.356,Y 33.471,Z 54.883,A 180.000,B 0.000,C 180.000} C_DIS
LIN {X 43.418,Y 33.615,Z 54.878,A 180.000,B 0.000,C 180.000} C_DIS
LIN {X 43.480,Y 33.760,Z 54.873,A 180.000,B 0.000,C 180.000} C_DIS
LIN {X 43.533,Y 33.908,Z 54.869,A 180.000,B 0.000,C 180.000} C_DIS
LIN {X 43.586,Y 34.057,Z 54.864,A 180.000,B 0.000,C 180.000} C_DIS
LIN {X 43.638,Y 34.205,Z 54.859,A 180.000,B 0.000,C 180.000} C_DIS
LIN {X 43.682,Y 34.357,Z 54.854,A 180.000,B 0.000,C 180.000} C_DIS
LIN {X 43.704,Y 34.432,Z 54.851,A 180.000,B 0.000,C 180.000} C_DIS
LIN {X 43.726,Y 34.508,Z 54.849,A 180.000,B 0.000,C 180.000} C_DIS
LIN {X 43.748,Y 34.583,Z 54.846,A 180.000,B 0.000,C 180.000} C_DIS
LIN {X 43.769,Y 34.659,Z 54.844,A 180.000,B 0.000,C 180.000} C_DIS
LIN {X 43.786,Y 34.736,Z 54.841,A 180.000,B 0.000,C 180.000} C_DIS
LIN {X 43.803,Y 34.813,Z 54.839,A 180.000,B 0.000,C 180.000} C_DIS
LIN {X 43.820,Y 34.890,Z 54.836,A 180.000,B 0.000,C 180.000} C_DIS
LIN {X 43.855,Y 35.044,Z 54.831,A 180.000,B 0.000,C 180.000} C_DIS
LIN {X 43.870,Y 35.121,Z 54.828,A 180.000,B 0.000,C 180.000} C_DIS
LIN {X 43.895,Y 35.277,Z 54.823,A 180.000,B 0.000,C 180.000} C_DIS
LIN {X 43.919,Y 35.432,Z 54.817,A 180.000,B 0.000,C 180.000} C_DIS
LIN {X 43.932,Y 35.510,Z 54.815,A 180.000,B 0.000,C 180.000} C_DIS
LIN {X 43.942,Y 35.588,Z 54.812,A 180.000,B 0.000,C 180.000} C_DIS
LIN {X 43.972,Y 35.902,Z 54.801,A 180.000,B 0.000,C 180.000} C_DIS
LIN {X 43.979,Y 35.980,Z 54.798,A 180.000,B 0.000,C 180.000} C_DIS
LIN {X 43.985,Y 36.058,Z 54.796,A 180.000,B 0.000,C 180.000} C_DIS
LIN {X 43.990,Y 36.216,Z 54.790,A 180.000,B 0.000,C 180.000} C_DIS
LIN {X 43.997,Y 36.452,Z 54.782,A 180.000,B 0.000,C 180.000} C_DIS
LIN {X 43.998,Y 36.531,Z 54.779,A 180.000,B 0.000,C 180.000} C_DIS
LIN {X 43.990,Y 36.767,Z 54.771,A 180.000,B 0.000,C 180.000} C_DIS
LIN {X 43.985,Y 36.924,Z 54.765,A 180.000,B 0.000,C 180.000} C_DIS
LIN {X 43.981,Y 37.003,Z 54.763,A 180.000,B 0.000,C 180.000} C_DIS
LIN {X 43.966,Y 37.160,Z 54.757,A 180.000,B 0.000,C 180.000} C_DIS
LIN {X 43.944,Y 37.395,Z 54.749,A 180.000,B 0.000,C 180.000} C_DIS
LIN {X 43.934,Y 37.473,Z 54.746,A 180.000,B 0.000,C 180.000} C_DIS
LIN {X 43.873,Y 37.862,Z 54.732,A 180.000,B 0.000,C 180.000} C_DIS
LIN {X 43.858,Y 37.939,Z 54.730,A 180.000,B 0.000,C 180.000} C_DIS
LIN {X 43.824,Y 38.093,Z 54.724,A 180.000,B 0.000,C 180.000} C_DIS
LIN {X 43.772,Y 38.324,Z 54.716,A 180.000,B 0.000,C 180.000} C_DIS
LIN {X 43.753,Y 38.400,Z 54.713,A 180.000,B 0.000,C 180.000} C_DIS
LIN {X 43.643,Y 38.778,Z 54.699,A 180.000,B 0.000,C 180.000} C_DIS
LIN {X 43.619,Y 38.853,Z 54.697,A 180.000,B 0.000,C 180.000} C_DIS
LIN {X 43.565,Y 39.001,Z 54.691,A 180.000,B 0.000,C 180.000} C_DIS
LIN {X 43.485,Y 39.224,Z 54.683,A 180.000,B 0.000,C 180.000} C_DIS
LIN {X 43.456,Y 39.297,Z 54.680,A 180.000,B 0.000,C 180.000} C_DIS
LIN {X 43.300,Y 39.658,Z 54.666,A 180.000,B 0.000,C 180.000} C_DIS
LIN {X 43.266,Y 39.729,Z 54.664,A 180.000,B 0.000,C 180.000} C_DIS
LIN {X 43.159,Y 39.940,Z 54.655,A 180.000,B 0.000,C 180.000} C_DIS
LIN {X 43.088,Y 40.080,Z 54.650,A 180.000,B 0.000,C 180.000} C_DIS
LIN {X 43.050,Y 40.149,Z 54.647,A 180.000,B 0.000,C 180.000} C_DIS
LIN {X 42.849,Y 40.488,Z 54.633,A 180.000,B 0.000,C 180.000} C_DIS
LIN {X 42.807,Y 40.554,Z 54.631,A 180.000,B 0.000,C 180.000} C_DIS
LIN {X 42.674,Y 40.750,Z 54.622,A 180.000,B 0.000,C 180.000} C_DIS
LIN {X 42.585,Y 40.880,Z 54.617,A 180.000,B 0.000,C 180.000} C_DIS
LIN {X 42.539,Y 40.944,Z 54.614,A 180.000,B 0.000,C 180.000} C_DIS
LIN {X 42.297,Y 41.255,Z 54.600,A 180.000,B 0.000,C 180.000} C_DIS
LIN {X 42.247,Y 41.315,Z 54.598,A 180.000,B 0.000,C 180.000} C_DIS
LIN {X 42.091,Y 41.492,Z 54.589,A 180.000,B 0.000,C 180.000} C_DIS
LIN {X 41.986,Y 41.610,Z 54.584,A 180.000,B 0.000,C 180.000} C_DIS
LIN {X 41.932,Y 41.668,Z 54.581,A 180.000,B 0.000,C 180.000} C_DIS
LIN {X 41.654,Y 41.946,Z 54.567,A 180.000,B 0.000,C 180.000} C_DIS
LIN {X 41.596,Y 41.999,Z 54.565,A 180.000,B 0.000,C 180.000} C_DIS
LIN {X 41.300,Y 42.260,Z 54.551,A 180.000,B 0.000,C 180.000} C_DIS
LIN {X 41.239,Y 42.309,Z 54.548,A 180.000,B 0.000,C 180.000} C_DIS
LIN {X 40.928,Y 42.551,Z 54.534,A 180.000,B 0.000,C 180.000} C_DIS
LIN {X 40.864,Y 42.596,Z 54.532,A 180.000,B 0.000,C 180.000} C_DIS
LIN {X 40.538,Y 42.818,Z 54.518,A 180.000,B 0.000,C 180.000} C_DIS
LIN {X 40.471,Y 42.859,Z 54.515,A 180.000,B 0.000,C 180.000} C_DIS
LIN {X 40.132,Y 43.060,Z 54.501,A 180.000,B 0.000,C 180.000} C_DIS
LIN {X 40.063,Y 43.097,Z 54.499,A 180.000,B 0.000,C 180.000} C_DIS
LIN {X 39.712,Y 43.275,Z 54.485,A 180.000,B 0.000,C 180.000} C_DIS
LIN {X 39.640,Y 43.308,Z 54.482,A 180.000,B 0.000,C 180.000} C_DIS
LIN {X 39.279,Y 43.464,Z 54.468,A 180.000,B 0.000,C 180.000} C_DIS
LIN {X 39.205,Y 43.492,Z 54.466,A 180.000,B 0.000,C 180.000} C_DIS
LIN {X 38.835,Y 43.625,Z 54.452,A 180.000,B 0.000,C 180.000} C_DIS
LIN {X 38.759,Y 43.649,Z 54.449,A 180.000,B 0.000,C 180.000} C_DIS
LIN {X 38.381,Y 43.758,Z 54.435,A 180.000,B 0.000,C 180.000} C_DIS
LIN {X 38.305,Y 43.777,Z 54.433,A 180.000,B 0.000,C 180.000} C_DIS
LIN {X 37.920,Y 43.863,Z 54.419,A 180.000,B 0.000,C 180.000} C_DIS
LIN {X 37.843,Y 43.876,Z 54.416,A 180.000,B 0.000,C 180.000} C_DIS
LIN {X 37.454,Y 43.937,Z 54.402,A 180.000,B 0.000,C 180.000} C_DIS
LIN {X 37.376,Y 43.946,Z 54.400,A 180.000,B 0.000,C 180.000} C_DIS
LIN {X 37.140,Y 43.968,Z 54.391,A 180.000,B 0.000,C 180.000} C_DIS
LIN {X 36.984,Y 43.983,Z 54.386,A 180.000,B 0.000,C 180.000} C_DIS
LIN {X 36.905,Y 43.986,Z 54.383,A 180.000,B 0.000,C 180.000} C_DIS
LIN {X 36.511,Y 43.998,Z 54.369,A 180.000,B 0.000,C 180.000} C_DIS
LIN {X 36.433,Y 43.997,Z 54.367,A 180.000,B 0.000,C 180.000} C_DIS
LIN {X 36.196,Y 43.989,Z 54.358,A 180.000,B 0.000,C 180.000} C_DIS
LIN {X 36.039,Y 43.984,Z 54.353,A 180.000,B 0.000,C 180.000} C_DIS
LIN {X 35.960,Y 43.977,Z 54.350,A 180.000,B 0.000,C 180.000} C_DIS
LIN {X 35.569,Y 43.940,Z 54.336,A 180.000,B 0.000,C 180.000} C_DIS
LIN {X 35.491,Y 43.929,Z 54.334,A 180.000,B 0.000,C 180.000} C_DIS
LIN {X 35.335,Y 43.904,Z 54.328,A 180.000,B 0.000,C 180.000} C_DIS
LIN {X 35.102,Y 43.867,Z 54.320,A 180.000,B 0.000,C 180.000} C_DIS
LIN {X 35.025,Y 43.850,Z 54.317,A 180.000,B 0.000,C 180.000} C_DIS
LIN {X 34.640,Y 43.764,Z 54.303,A 180.000,B 0.000,C 180.000} C_DIS
LIN {X 34.565,Y 43.743,Z 54.301,A 180.000,B 0.000,C 180.000} C_DIS
LIN {X 34.413,Y 43.699,Z 54.295,A 180.000,B 0.000,C 180.000} C_DIS
LIN {X 34.187,Y 43.633,Z 54.287,A 180.000,B 0.000,C 180.000} C_DIS
LIN {X 34.112,Y 43.606,Z 54.284,A 180.000,B 0.000,C 180.000} C_DIS
LIN {X 33.890,Y 43.526,Z 54.276,A 180.000,B 0.000,C 180.000} C_DIS
LIN {X 33.742,Y 43.473,Z 54.270,A 180.000,B 0.000,C 180.000} C_DIS
LIN {X 33.669,Y 43.442,Z 54.268,A 180.000,B 0.000,C 180.000} C_DIS
LIN {X 33.525,Y 43.379,Z 54.262,A 180.000,B 0.000,C 180.000} C_DIS
LIN {X 33.308,Y 43.285,Z 54.254,A 180.000,B 0.000,C 180.000} C_DIS
LIN {X 33.238,Y 43.250,Z 54.251,A 180.000,B 0.000,C 180.000} C_DIS
LIN {X 33.027,Y 43.143,Z 54.243,A 180.000,B 0.000,C 180.000} C_DIS
LIN {X 32.957,Y 43.107,Z 54.240,A 180.000,B 0.000,C 180.000} C_DIS
LIN {X 32.887,Y 43.071,Z 54.237,A 180.000,B 0.000,C 180.000} C_DIS
LIN {X 32.819,Y 43.031,Z 54.235,A 180.000,B 0.000,C 180.000} C_DIS
LIN {X 32.684,Y 42.951,Z 54.229,A 180.000,B 0.000,C 180.000} C_DIS
LIN {X 32.548,Y 42.871,Z 54.224,A 180.000,B 0.000,C 180.000} C_DIS
LIN {X 32.480,Y 42.830,Z 54.221,A 180.000,B 0.000,C 180.000} C_DIS
LIN {X 32.350,Y 42.742,Z 54.215,A 180.000,B 0.000,C 180.000} C_DIS
LIN {X 32.285,Y 42.698,Z 54.213,A 180.000,B 0.000,C 180.000} C_DIS
LIN {X 32.155,Y 42.609,Z 54.207,A 180.000,B 0.000,C 180.000} C_DIS
LIN {X 32.090,Y 42.565,Z 54.204,A 180.000,B 0.000,C 180.000} C_DIS
LIN {X 32.027,Y 42.516,Z 54.202,A 180.000,B 0.000,C 180.000} C_DIS
LIN {X 31.903,Y 42.420,Z 54.196,A 180.000,B 0.000,C 180.000} C_DIS
LIN {X 31.778,Y 42.323,Z 54.191,A 180.000,B 0.000,C 180.000} C_DIS
LIN {X 31.716,Y 42.275,Z 54.188,A 180.000,B 0.000,C 180.000} C_DIS
LIN {X 31.598,Y 42.170,Z 54.182,A 180.000,B 0.000,C 180.000} C_DIS
LIN {X 31.480,Y 42.066,Z 54.177,A 180.000,B 0.000,C 180.000} C_DIS
LIN {X 31.421,Y 42.014,Z 54.174,A 180.000,B 0.000,C 180.000} C_DIS
LIN {X 31.362,Y 41.962,Z 54.172,A 180.000,B 0.000,C 180.000} C_DIS
LIN {X 31.251,Y 41.850,Z 54.166,A 180.000,B 0.000,C 180.000} C_DIS
LIN {X 31.195,Y 41.795,Z 54.164,A 180.000,B 0.000,C 180.000} C_DIS
LIN {X 31.139,Y 41.739,Z 54.161,A 180.000,B 0.000,C 180.000} C_DIS
LIN {X 31.084,Y 41.683,Z 54.159,A 180.000,B 0.000,C 180.000} C_DIS
LIN {X 31.028,Y 41.627,Z 54.156,A 180.000,B 0.000,C 180.000} C_DIS
LIN {X 30.924,Y 41.509,Z 54.151,A 180.000,B 0.000,C 180.000} C_DIS
LIN {X 30.872,Y 41.450,Z 54.149,A 180.000,B 0.000,C 180.000} C_DIS
LIN {X 30.768,Y 41.332,Z 54.144,A 180.000,B 0.000,C 180.000} C_DIS
LIN {X 30.668,Y 41.210,Z 54.139,A 180.000,B 0.000,C 180.000} C_DIS
LIN {X 30.572,Y 41.086,Z 54.134,A 180.000,B 0.000,C 180.000} C_DIS
LIN {X 30.475,Y 40.961,Z 54.129,A 180.000,B 0.000,C 180.000} C_DIS
LIN {X 30.383,Y 40.834,Z 54.124,A 180.000,B 0.000,C 180.000} C_DIS
LIN {X 30.294,Y 40.703,Z 54.120,A 180.000,B 0.000,C 180.000} C_DIS
LIN {X 30.206,Y 40.573,Z 54.115,A 180.000,B 0.000,C 180.000} C_DIS
LIN {X 30.122,Y 40.440,Z 54.111,A 180.000,B 0.000,C 180.000} C_DIS
LIN {X 30.042,Y 40.304,Z 54.106,A 180.000,B 0.000,C 180.000} C_DIS
LIN {X 29.962,Y 40.168,Z 54.102,A 180.000,B 0.000,C 180.000} C_DIS
LIN {X 29.887,Y 40.030,Z 54.097,A 180.000,B 0.000,C 180.000} C_DIS
LIN {X 29.815,Y 39.890,Z 54.093,A 180.000,B 0.000,C 180.000} C_DIS
LIN {X 29.744,Y 39.749,Z 54.089,A 180.000,B 0.000,C 180.000} C_DIS
LIN {X 29.678,Y 39.607,Z 54.085,A 180.000,B 0.000,C 180.000} C_DIS
LIN {X 29.615,Y 39.462,Z 54.081,A 180.000,B 0.000,C 180.000} C_DIS
LIN {X 29.552,Y 39.317,Z 54.077,A 180.000,B 0.000,C 180.000} C_DIS
LIN {X 29.495,Y 39.171,Z 54.073,A 180.000,B 0.000,C 180.000} C_DIS
LIN {X 29.442,Y 39.022,Z 54.070,A 180.000,B 0.000,C 180.000} C_DIS
LIN {X 29.389,Y 38.874,Z 54.066,A 180.000,B 0.000,C 180.000} C_DIS
LIN {X 29.341,Y 38.724,Z 54.062,A 180.000,B 0.000,C 180.000} C_DIS
LIN {X 29.297,Y 38.573,Z 54.059,A 180.000,B 0.000,C 180.000} C_DIS
LIN {X 29.253,Y 38.422,Z 54.056,A 180.000,B 0.000,C 180.000} C_DIS
LIN {X 29.215,Y 38.269,Z 54.052,A 180.000,B 0.000,C 180.000} C_DIS
LIN {X 29.181,Y 38.115,Z 54.049,A 180.000,B 0.000,C 180.000} C_DIS
LIN {X 29.147,Y 37.961,Z 54.046,A 180.000,B 0.000,C 180.000} C_DIS
LIN {X 29.118,Y 37.806,Z 54.043,A 180.000,B 0.000,C 180.000} C_DIS
LIN {X 29.094,Y 37.651,Z 54.040,A 180.000,B 0.000,C 180.000} C_DIS
LIN {X 29.069,Y 37.495,Z 54.037,A 180.000,B 0.000,C 180.000} C_DIS
LIN {X 29.051,Y 37.339,Z 54.034,A 180.000,B 0.000,C 180.000} C_DIS
LIN {X 29.036,Y 37.182,Z 54.032,A 180.000,B 0.000,C 180.000} C_DIS
LIN {X 29.021,Y 37.025,Z 54.029,A 180.000,B 0.000,C 180.000} C_DIS
LIN {X 29.013,Y 36.868,Z 54.027,A 180.000,B 0.000,C 180.000} C_DIS
LIN {X 29.003,Y 36.553,Z 54.022,A 180.000,B 0.000,C 180.000} C_DIS
LIN {X 29.009,Y 36.238,Z 54.018,A 180.000,B 0.000,C 180.000} C_DIS
LIN {X 29.026,Y 35.924,Z 54.014,A 180.000,B 0.000,C 180.000} C_DIS
LIN {X 29.056,Y 35.610,Z 54.011,A 180.000,B 0.000,C 180.000} C_DIS
LIN {X 29.102,Y 35.299,Z 54.008,A 180.000,B 0.000,C 180.000} C_DIS
LIN {X 29.158,Y 34.989,Z 54.005,A 180.000,B 0.000,C 180.000} C_DIS
LIN {X 29.226,Y 34.681,Z 54.003,A 180.000,B 0.000,C 180.000} C_DIS
LIN {X 29.312,Y 34.378,Z 54.002,A 180.000,B 0.000,C 180.000} C_DIS
LIN {X 29.406,Y 34.078,Z 54.001,A 180.000,B 0.000,C 180.000} C_DIS
LIN {X 29.513,Y 33.781,Z 54.000,A 180.000,B 0.000,C 180.000} C_DIS
LIN {X 29.603,Y 33.566,Z 54.000,A 180.000,B 0.000,C 180.000} C_DIS
; Cutting Move Starts
LIN {X 29.679,Y 33.390,Z 54.000,A 180.000,B 0.000,C 180.000} C_DIS
LIN {X 29.742,Y 33.254,Z 54.000,A 180.000,B 0.000,C 180.000} C_DIS
LIN {X 29.924,Y 32.897,Z 54.000,A 180.000,B 0.000,C 180.000} C_DIS
LIN {X 30.029,Y 32.718,Z 54.000,A 180.000,B 0.000,C 180.000} C_DIS
LIN {X 30.135,Y 32.539,Z 54.000,A 180.000,B 0.000,C 180.000} C_DIS
LIN {X 30.215,Y 32.413,Z 54.000,A 180.000,B 0.000,C 180.000} C_DIS
LIN {X 30.394,Y 32.150,Z 54.000,A 180.000,B 0.000,C 180.000} C_DIS
LIN {X 30.503,Y 32.003,Z 54.000,A 180.000,B 0.000,C 180.000} C_DIS
LIN {X 30.641,Y 31.824,Z 54.000,A 180.000,B 0.000,C 180.000} C_DIS
LIN {X 30.752,Y 31.687,Z 54.000,A 180.000,B 0.000,C 180.000} C_DIS
LIN {X 30.945,Y 31.467,Z 54.000,A 180.000,B 0.000,C 180.000} C_DIS
LIN {X 31.109,Y 31.291,Z 54.000,A 180.000,B 0.000,C 180.000} C_DIS
LIN {X 31.291,Y 31.109,Z 54.000,A 180.000,B 0.000,C 180.000} C_DIS
LIN {X 31.467,Y 30.945,Z 54.000,A 180.000,B 0.000,C 180.000} C_DIS
LIN {X 31.687,Y 30.752,Z 54.000,A 180.000,B 0.000,C 180.000} C_DIS
LIN {X 31.824,Y 30.641,Z 54.000,A 180.000,B 0.000,C 180.000} C_DIS
LIN {X 32.003,Y 30.503,Z 54.000,A 180.000,B 0.000,C 180.000} C_DIS
LIN {X 32.150,Y 30.394,Z 54.000,A 180.000,B 0.000,C 180.000} C_DIS
LIN {X 32.413,Y 30.215,Z 54.000,A 180.000,B 0.000,C 180.000} C_DIS
LIN {X 32.539,Y 30.135,Z 54.000,A 180.000,B 0.000,C 180.000} C_DIS
LIN {X 32.718,Y 30.029,Z 54.000,A 180.000,B 0.000,C 180.000} C_DIS
LIN {X 32.897,Y 29.924,Z 54.000,A 180.000,B 0.000,C 180.000} C_DIS
LIN {X 33.254,Y 29.742,Z 54.000,A 180.000,B 0.000,C 180.000} C_DIS
LIN {X 33.390,Y 29.679,Z 54.000,A 180.000,B 0.000,C 180.000} C_DIS
LIN {X 33.612,Y 29.583,Z 54.000,A 180.000,B 0.000,C 180.000} C_DIS
LIN {X 33.791,Y 29.509,Z 54.000,A 180.000,B 0.000,C 180.000} C_DIS
LIN {X 34.148,Y 29.381,Z 54.000,A 180.000,B 0.000,C 180.000} C_DIS
LIN {X 34.327,Y 29.326,Z 54.000,A 180.000,B 0.000,C 180.000} C_DIS
LIN {X 34.506,Y 29.274,Z 54.000,A 180.000,B 0.000,C 180.000} C_DIS
LIN {X 34.685,Y 29.226,Z 54.000,A 180.000,B 0.000,C 180.000} C_DIS
LIN {X 35.056,Y 29.143,Z 54.000,A 180.000,B 0.000,C 180.000} C_DIS
LIN {X 35.221,Y 29.114,Z 54.000,A 180.000,B 0.000,C 180.000} C_DIS
LIN {X 35.400,Y 29.086,Z 54.000,A 180.000,B 0.000,C 180.000} C_DIS
LIN {X 35.578,Y 29.059,Z 54.000,A 180.000,B 0.000,C 180.000} C_DIS
LIN {X 35.936,Y 29.025,Z 54.000,A 180.000,B 0.000,C 180.000} C_DIS
LIN {X 36.115,Y 29.013,Z 54.000,A 180.000,B 0.000,C 180.000} C_DIS
LIN {X 36.472,Y 29.002,Z 54.000,A 180.000,B 0.000,C 180.000} C_DIS
LIN {X 36.651,Y 29.006,Z 54.000,A 180.000,B 0.000,C 180.000} C_DIS
LIN {X 36.830,Y 29.012,Z 54.000,A 180.000,B 0.000,C 180.000} C_DIS
LIN {X 37.009,Y 29.020,Z 54.000,A 180.000,B 0.000,C 180.000} C_DIS
LIN {X 37.366,Y 29.053,Z 54.000,A 180.000,B 0.000,C 180.000} C_DIS
LIN {X 37.545,Y 29.077,Z 54.000,A 180.000,B 0.000,C 180.000} C_DIS
LIN {X 37.748,Y 29.109,Z 54.000,A 180.000,B 0.000,C 180.000} C_DIS
LIN {X 37.902,Y 29.134,Z 54.000,A 180.000,B 0.000,C 180.000} C_DIS
LIN {X 37.944,Y 29.143,Z 54.000,A 180.000,B 0.000,C 180.000} C_DIS
LIN {X 38.260,Y 29.213,Z 54.000,A 180.000,B 0.000,C 180.000} C_DIS
LIN {X 38.439,Y 29.258,Z 54.000,A 180.000,B 0.000,C 180.000} C_DIS
LIN {X 38.796,Y 29.362,Z 54.000,A 180.000,B 0.000,C 180.000} C_DIS
LIN {X 38.975,Y 29.425,Z 54.000,A 180.000,B 0.000,C 180.000} C_DIS
LIN {X 39.184,Y 29.500,Z 54.000,A 180.000,B 0.000,C 180.000} C_DIS
LIN {X 39.333,Y 29.559,Z 54.000,A 180.000,B 0.000,C 180.000} C_DIS
LIN {X 39.690,Y 29.714,Z 54.000,A 180.000,B 0.000,C 180.000} C_DIS
LIN {X 39.869,Y 29.805,Z 54.000,A 180.000,B 0.000,C 180.000} C_DIS
LIN {X 40.048,Y 29.896,Z 54.000,A 180.000,B 0.000,C 180.000} C_DIS
LIN {X 40.226,Y 29.996,Z 54.000,A 180.000,B 0.000,C 180.000} C_DIS
LIN {X 40.405,Y 30.102,Z 54.000,A 180.000,B 0.000,C 180.000} C_DIS
LIN {X 40.584,Y 30.213,Z 54.000,A 180.000,B 0.000,C 180.000} C_DIS
LIN {X 40.850,Y 30.394,Z 54.000,A 180.000,B 0.000,C 180.000} C_DIS
LIN {X 40.942,Y 30.460,Z 54.000,A 180.000,B 0.000,C 180.000} C_DIS
LIN {X 41.120,Y 30.598,Z 54.000,A 180.000,B 0.000,C 180.000} C_DIS
LIN {X 41.299,Y 30.739,Z 54.000,A 180.000,B 0.000,C 180.000} C_DIS
LIN {X 41.516,Y 30.930,Z 54.000,A 180.000,B 0.000,C 180.000} C_DIS
LIN {X 41.657,Y 31.057,Z 54.000,A 180.000,B 0.000,C 180.000} C_DIS
LIN {X 41.888,Y 31.288,Z 54.000,A 180.000,B 0.000,C 180.000} C_DIS
LIN {X 42.014,Y 31.421,Z 54.000,A 180.000,B 0.000,C 180.000} C_DIS
LIN {X 42.212,Y 31.646,Z 54.000,A 180.000,B 0.000,C 180.000} C_DIS
LIN {X 42.359,Y 31.824,Z 54.000,A 180.000,B 0.000,C 180.000} C_DIS
LIN {X 42.550,Y 32.072,Z 54.000,A 180.000,B 0.000,C 180.000} C_DIS
LIN {X 42.627,Y 32.182,Z 54.000,A 180.000,B 0.000,C 180.000} C_DIS
LIN {X 42.749,Y 32.361,Z 54.000,A 180.000,B 0.000,C 180.000} C_DIS
LIN {X 42.865,Y 32.539,Z 54.000,A 180.000,B 0.000,C 180.000} C_DIS
LIN {X 42.971,Y 32.718,Z 54.000,A 180.000,B 0.000,C 180.000} C_DIS
LIN {X 43.076,Y 32.897,Z 54.000,A 180.000,B 0.000,C 180.000} C_DIS
LIN {X 43.266,Y 33.269,Z 54.000,A 180.000,B 0.000,C 180.000} C_DIS
LIN {X 43.340,Y 33.433,Z 54.000,A 180.000,B 0.000,C 180.000} C_DIS
LIN {X 43.444,Y 33.675,Z 54.000,A 180.000,B 0.000,C 180.000} C_DIS
LIN {X 43.491,Y 33.791,Z 54.000,A 180.000,B 0.000,C 180.000} C_DIS
LIN {X 43.623,Y 34.159,Z 54.000,A 180.000,B 0.000,C 180.000} C_DIS
LIN {X 43.674,Y 34.327,Z 54.000,A 180.000,B 0.000,C 180.000} C_DIS
LIN {X 43.726,Y 34.506,Z 54.000,A 180.000,B 0.000,C 180.000} C_DIS
LIN {X 43.774,Y 34.685,Z 54.000,A 180.000,B 0.000,C 180.000} C_DIS
LIN {X 43.854,Y 35.042,Z 54.000,A 180.000,B 0.000,C 180.000} C_DIS
LIN {X 43.886,Y 35.221,Z 54.000,A 180.000,B 0.000,C 180.000} C_DIS
LIN {X 43.914,Y 35.400,Z 54.000,A 180.000,B 0.000,C 180.000} C_DIS
LIN {X 43.941,Y 35.578,Z 54.000,A 180.000,B 0.000,C 180.000} C_DIS
LIN {X 43.981,Y 35.994,Z 54.000,A 180.000,B 0.000,C 180.000} C_DIS
LIN {X 43.987,Y 36.115,Z 54.000,A 180.000,B 0.000,C 180.000} C_DIS
LIN {X 43.998,Y 36.472,Z 54.000,A 180.000,B 0.000,C 180.000} C_DIS
LIN {X 43.994,Y 36.651,Z 54.000,A 180.000,B 0.000,C 180.000} C_DIS
LIN {X 43.988,Y 36.830,Z 54.000,A 180.000,B 0.000,C 180.000} C_DIS
LIN {X 43.981,Y 37.006,Z 54.000,A 180.000,B 0.000,C 180.000} C_DIS
LIN {X 43.947,Y 37.366,Z 54.000,A 180.000,B 0.000,C 180.000} C_DIS
LIN {X 43.923,Y 37.545,Z 54.000,A 180.000,B 0.000,C 180.000} C_DIS
LIN {X 43.866,Y 37.902,Z 54.000,A 180.000,B 0.000,C 180.000} C_DIS
LIN {X 43.827,Y 38.081,Z 54.000,A 180.000,B 0.000,C 180.000} C_DIS
LIN {X 43.787,Y 38.260,Z 54.000,A 180.000,B 0.000,C 180.000} C_DIS
LIN {X 43.742,Y 38.439,Z 54.000,A 180.000,B 0.000,C 180.000} C_DIS
LIN {X 43.638,Y 38.796,Z 54.000,A 180.000,B 0.000,C 180.000} C_DIS
LIN {X 43.623,Y 38.841,Z 54.000,A 180.000,B 0.000,C 180.000} C_DIS
LIN {X 43.511,Y 39.154,Z 54.000,A 180.000,B 0.000,C 180.000} C_DIS
LIN {X 43.444,Y 39.325,Z 54.000,A 180.000,B 0.000,C 180.000} C_DIS
LIN {X 43.286,Y 39.690,Z 54.000,A 180.000,B 0.000,C 180.000} C_DIS
LIN {X 43.266,Y 39.731,Z 54.000,A 180.000,B 0.000,C 180.000} C_DIS
LIN {X 43.087,Y 40.082,Z 54.000,A 180.000,B 0.000,C 180.000} C_DIS
LIN {X 43.004,Y 40.226,Z 54.000,A 180.000,B 0.000,C 180.000} C_DIS
LIN {X 42.898,Y 40.405,Z 54.000,A 180.000,B 0.000,C 180.000} C_DIS
LIN {X 42.787,Y 40.584,Z 54.000,A 180.000,B 0.000,C 180.000} C_DIS
LIN {X 42.665,Y 40.763,Z 54.000,A 180.000,B 0.000,C 180.000} C_DIS
LIN {X 42.550,Y 40.928,Z 54.000,A 180.000,B 0.000,C 180.000} C_DIS
LIN {X 42.372,Y 41.159,Z 54.000,A 180.000,B 0.000,C 180.000} C_DIS
LIN {X 42.261,Y 41.299,Z 54.000,A 180.000,B 0.000,C 180.000} C_DIS
LIN {X 42.014,Y 41.579,Z 54.000,A 180.000,B 0.000,C 180.000} C_DIS
LIN {X 41.943,Y 41.657,Z 54.000,A 180.000,B 0.000,C 180.000} C_DIS
LIN {X 41.657,Y 41.943,Z 54.000,A 180.000,B 0.000,C 180.000} C_DIS
LIN {X 41.579,Y 42.014,Z 54.000,A 180.000,B 0.000,C 180.000} C_DIS
LIN {X 41.299,Y 42.261,Z 54.000,A 180.000,B 0.000,C 180.000} C_DIS
LIN {X 41.159,Y 42.372,Z 54.000,A 180.000,B 0.000,C 180.000} C_DIS
LIN {X 40.928,Y 42.550,Z 54.000,A 180.000,B 0.000,C 180.000} C_DIS
LIN {X 40.763,Y 42.665,Z 54.000,A 180.000,B 0.000,C 180.000} C_DIS
LIN {X 40.584,Y 42.787,Z 54.000,A 180.000,B 0.000,C 180.000} C_DIS
LIN {X 40.405,Y 42.898,Z 54.000,A 180.000,B 0.000,C 180.000} C_DIS
LIN {X 40.226,Y 43.004,Z 54.000,A 180.000,B 0.000,C 180.000} C_DIS
LIN {X 40.082,Y 43.087,Z 54.000,A 180.000,B 0.000,C 180.000} C_DIS
LIN {X 39.731,Y 43.266,Z 54.000,A 180.000,B 0.000,C 180.000} C_DIS
LIN {X 39.690,Y 43.286,Z 54.000,A 180.000,B 0.000,C 180.000} C_DIS
LIN {X 39.325,Y 43.444,Z 54.000,A 180.000,B 0.000,C 180.000} C_DIS
LIN {X 39.154,Y 43.511,Z 54.000,A 180.000,B 0.000,C 180.000} C_DIS
LIN {X 38.841,Y 43.623,Z 54.000,A 180.000,B 0.000,C 180.000} C_DIS
LIN {X 38.796,Y 43.638,Z 54.000,A 180.000,B 0.000,C 180.000} C_DIS
LIN {X 38.439,Y 43.742,Z 54.000,A 180.000,B 0.000,C 180.000} C_DIS
LIN {X 38.260,Y 43.787,Z 54.000,A 180.000,B 0.000,C 180.000} C_DIS
LIN {X 38.081,Y 43.827,Z 54.000,A 180.000,B 0.000,C 180.000} C_DIS
LIN {X 37.902,Y 43.866,Z 54.000,A 180.000,B 0.000,C 180.000} C_DIS
LIN {X 37.545,Y 43.923,Z 54.000,A 180.000,B 0.000,C 180.000} C_DIS
LIN {X 37.366,Y 43.947,Z 54.000,A 180.000,B 0.000,C 180.000} C_DIS
LIN {X 37.006,Y 43.981,Z 54.000,A 180.000,B 0.000,C 180.000} C_DIS
LIN {X 36.830,Y 43.988,Z 54.000,A 180.000,B 0.000,C 180.000} C_DIS
LIN {X 36.651,Y 43.994,Z 54.000,A 180.000,B 0.000,C 180.000} C_DIS
LIN {X 36.472,Y 43.998,Z 54.000,A 180.000,B 0.000,C 180.000} C_DIS
LIN {X 36.115,Y 43.987,Z 54.000,A 180.000,B 0.000,C 180.000} C_DIS
LIN {X 35.994,Y 43.981,Z 54.000,A 180.000,B 0.000,C 180.000} C_DIS
LIN {X 35.578,Y 43.941,Z 54.000,A 180.000,B 0.000,C 180.000} C_DIS
LIN {X 35.400,Y 43.914,Z 54.000,A 180.000,B 0.000,C 180.000} C_DIS
LIN {X 35.221,Y 43.886,Z 54.000,A 180.000,B 0.000,C 180.000} C_DIS
LIN {X 35.042,Y 43.854,Z 54.000,A 180.000,B 0.000,C 180.000} C_DIS
LIN {X 34.685,Y 43.774,Z 54.000,A 180.000,B 0.000,C 180.000} C_DIS
LIN {X 34.506,Y 43.726,Z 54.000,A 180.000,B 0.000,C 180.000} C_DIS
LIN {X 34.327,Y 43.674,Z 54.000,A 180.000,B 0.000,C 180.000} C_DIS
LIN {X 34.159,Y 43.623,Z 54.000,A 180.000,B 0.000,C 180.000} C_DIS
LIN {X 33.791,Y 43.491,Z 54.000,A 180.000,B 0.000,C 180.000} C_DIS
LIN {X 33.675,Y 43.444,Z 54.000,A 180.000,B 0.000,C 180.000} C_DIS
LIN {X 33.433,Y 43.340,Z 54.000,A 180.000,B 0.000,C 180.000} C_DIS
LIN {X 33.269,Y 43.266,Z 54.000,A 180.000,B 0.000,C 180.000} C_DIS
LIN {X 32.897,Y 43.076,Z 54.000,A 180.000,B 0.000,C 180.000} C_DIS
LIN {X 32.718,Y 42.971,Z 54.000,A 180.000,B 0.000,C 180.000} C_DIS
LIN {X 32.539,Y 42.865,Z 54.000,A 180.000,B 0.000,C 180.000} C_DIS
LIN {X 32.361,Y 42.749,Z 54.000,A 180.000,B 0.000,C 180.000} C_DIS
LIN {X 32.182,Y 42.627,Z 54.000,A 180.000,B 0.000,C 180.000} C_DIS
LIN {X 32.072,Y 42.550,Z 54.000,A 180.000,B 0.000,C 180.000} C_DIS
LIN {X 31.824,Y 42.359,Z 54.000,A 180.000,B 0.000,C 180.000} C_DIS
LIN {X 31.646,Y 42.212,Z 54.000,A 180.000,B 0.000,C 180.000} C_DIS
LIN {X 31.421,Y 42.014,Z 54.000,A 180.000,B 0.000,C 180.000} C_DIS
LIN {X 31.288,Y 41.888,Z 54.000,A 180.000,B 0.000,C 180.000} C_DIS
LIN {X 31.057,Y 41.657,Z 54.000,A 180.000,B 0.000,C 180.000} C_DIS
LIN {X 30.930,Y 41.516,Z 54.000,A 180.000,B 0.000,C 180.000} C_DIS
LIN {X 30.739,Y 41.299,Z 54.000,A 180.000,B 0.000,C 180.000} C_DIS
LIN {X 30.598,Y 41.120,Z 54.000,A 180.000,B 0.000,C 180.000} C_DIS
LIN {X 30.460,Y 40.942,Z 54.000,A 180.000,B 0.000,C 180.000} C_DIS
LIN {X 30.394,Y 40.850,Z 54.000,A 180.000,B 0.000,C 180.000} C_DIS
LIN {X 30.213,Y 40.584,Z 54.000,A 180.000,B 0.000,C 180.000} C_DIS
LIN {X 30.102,Y 40.405,Z 54.000,A 180.000,B 0.000,C 180.000} C_DIS
LIN {X 29.996,Y 40.226,Z 54.000,A 180.000,B 0.000,C 180.000} C_DIS
LIN {X 29.896,Y 40.048,Z 54.000,A 180.000,B 0.000,C 180.000} C_DIS
LIN {X 29.805,Y 39.869,Z 54.000,A 180.000,B 0.000,C 180.000} C_DIS
LIN {X 29.714,Y 39.690,Z 54.000,A 180.000,B 0.000,C 180.000} C_DIS
LIN {X 29.559,Y 39.333,Z 54.000,A 180.000,B 0.000,C 180.000} C_DIS
LIN {X 29.500,Y 39.184,Z 54.000,A 180.000,B 0.000,C 180.000} C_DIS
LIN {X 29.425,Y 38.975,Z 54.000,A 180.000,B 0.000,C 180.000} C_DIS
LIN {X 29.362,Y 38.796,Z 54.000,A 180.000,B 0.000,C 180.000} C_DIS
LIN {X 29.258,Y 38.439,Z 54.000,A 180.000,B 0.000,C 180.000} C_DIS
LIN {X 29.213,Y 38.260,Z 54.000,A 180.000,B 0.000,C 180.000} C_DIS
LIN {X 29.143,Y 37.944,Z 54.000,A 180.000,B 0.000,C 180.000} C_DIS
LIN {X 29.134,Y 37.902,Z 54.000,A 180.000,B 0.000,C 180.000} C_DIS
LIN {X 29.077,Y 37.545,Z 54.000,A 180.000,B 0.000,C 180.000} C_DIS
LIN {X 29.053,Y 37.366,Z 54.000,A 180.000,B 0.000,C 180.000} C_DIS
LIN {X 29.020,Y 37.009,Z 54.000,A 180.000,B 0.000,C 180.000} C_DIS
LIN {X 29.012,Y 36.830,Z 54.000,A 180.000,B 0.000,C 180.000} C_DIS
LIN {X 29.006,Y 36.651,Z 54.000,A 180.000,B 0.000,C 180.000} C_DIS
LIN {X 29.002,Y 36.472,Z 54.000,A 180.000,B 0.000,C 180.000} C_DIS
LIN {X 29.013,Y 36.115,Z 54.000,A 180.000,B 0.000,C 180.000} C_DIS
LIN {X 29.025,Y 35.936,Z 54.000,A 180.000,B 0.000,C 180.000} C_DIS
LIN {X 29.059,Y 35.578,Z 54.000,A 180.000,B 0.000,C 180.000} C_DIS
LIN {X 29.086,Y 35.400,Z 54.000,A 180.000,B 0.000,C 180.000} C_DIS
LIN {X 29.114,Y 35.221,Z 54.000,A 180.000,B 0.000,C 180.000} C_DIS
LIN {X 29.143,Y 35.056,Z 54.000,A 180.000,B 0.000,C 180.000} C_DIS
LIN {X 29.226,Y 34.685,Z 54.000,A 180.000,B 0.000,C 180.000} C_DIS
LIN {X 29.274,Y 34.506,Z 54.000,A 180.000,B 0.000,C 180.000} C_DIS
LIN {X 29.326,Y 34.327,Z 54.000,A 180.000,B 0.000,C 180.000} C_DIS
LIN {X 29.381,Y 34.148,Z 54.000,A 180.000,B 0.000,C 180.000} C_DIS
LIN {X 29.509,Y 33.791,Z 54.000,A 180.000,B 0.000,C 180.000} C_DIS
LIN {X 29.583,Y 33.612,Z 54.000,A 180.000,B 0.000,C 180.000} C_DIS
LIN {X 29.603,Y 33.566,Z 54.000,A 180.000,B 0.000,C 180.000} C_DIS
; Link Move Starts
LIN {X 29.730,Y 33.278,Z 54.000,A 180.000,B 0.000,C 180.000} C_DIS
LIN {X 29.873,Y 32.997,Z 53.999,A 180.000,B 0.000,C 180.000} C_DIS
LIN {X 30.026,Y 32.722,Z 53.998,A 180.000,B 0.000,C 180.000} C_DIS
LIN {X 30.189,Y 32.452,Z 53.996,A 180.000,B 0.000,C 180.000} C_DIS
LIN {X 30.366,Y 32.192,Z 53.994,A 180.000,B 0.000,C 180.000} C_DIS
LIN {X 30.553,Y 31.939,Z 53.991,A 180.000,B 0.000,C 180.000} C_DIS
LIN {X 30.748,Y 31.691,Z 53.988,A 180.000,B 0.000,C 180.000} C_DIS
LIN {X 30.956,Y 31.455,Z 53.985,A 180.000,B 0.000,C 180.000} C_DIS
LIN {X 31.173,Y 31.227,Z 53.981,A 180.000,B 0.000,C 180.000} C_DIS
LIN {X 31.398,Y 31.006,Z 53.977,A 180.000,B 0.000,C 180.000} C_DIS
LIN {X 31.634,Y 30.798,Z 53.972,A 180.000,B 0.000,C 180.000} C_DIS
LIN {X 31.754,Y 30.696,Z 53.969,A 180.000,B 0.000,C 180.000} C_DIS
LIN {X 31.879,Y 30.599,Z 53.967,A 180.000,B 0.000,C 180.000} C_DIS
LIN {X 32.003,Y 30.503,Z 53.964,A 180.000,B 0.000,C 180.000} C_DIS
LIN {X 32.129,Y 30.408,Z 53.961,A 180.000,B 0.000,C 180.000} C_DIS
LIN {X 32.260,Y 30.320,Z 53.959,A 180.000,B 0.000,C 180.000} C_DIS
LIN {X 32.390,Y 30.231,Z 53.956,A 180.000,B 0.000,C 180.000} C_DIS
LIN {X 32.522,Y 30.145,Z 53.952,A 180.000,B 0.000,C 180.000} C_DIS
LIN {X 32.657,Y 30.065,Z 53.949,A 180.000,B 0.000,C 180.000} C_DIS
LIN {X 32.793,Y 29.985,Z 53.946,A 180.000,B 0.000,C 180.000} C_DIS
LIN {X 32.930,Y 29.907,Z 53.943,A 180.000,B 0.000,C 180.000} C_DIS
LIN {X 33.070,Y 29.836,Z 53.939,A 180.000,B 0.000,C 180.000} C_DIS
LIN {X 33.211,Y 29.764,Z 53.936,A 180.000,B 0.000,C 180.000} C_DIS
LIN {X 33.352,Y 29.695,Z 53.932,A 180.000,B 0.000,C 180.000} C_DIS
LIN {X 33.497,Y 29.633,Z 53.928,A 180.000,B 0.000,C 180.000} C_DIS
LIN {X 33.641,Y 29.570,Z 53.925,A 180.000,B 0.000,C 180.000} C_DIS
LIN {X 33.787,Y 29.511,Z 53.921,A 180.000,B 0.000,C 180.000} C_DIS
LIN {X 33.935,Y 29.457,Z 53.917,A 180.000,B 0.000,C 180.000} C_DIS
LIN {X 34.083,Y 29.404,Z 53.913,A 180.000,B 0.000,C 180.000} C_DIS
LIN {X 34.233,Y 29.354,Z 53.909,A 180.000,B 0.000,C 180.000} C_DIS
LIN {X 34.384,Y 29.310,Z 53.905,A 180.000,B 0.000,C 180.000} C_DIS
LIN {X 34.535,Y 29.266,Z 53.900,A 180.000,B 0.000,C 180.000} C_DIS
LIN {X 34.687,Y 29.225,Z 53.896,A 180.000,B 0.000,C 180.000} C_DIS
LIN {X 34.841,Y 29.191,Z 53.892,A 180.000,B 0.000,C 180.000} C_DIS
LIN {X 34.995,Y 29.156,Z 53.887,A 180.000,B 0.000,C 180.000} C_DIS
LIN {X 35.149,Y 29.125,Z 53.883,A 180.000,B 0.000,C 180.000} C_DIS
LIN {X 35.305,Y 29.101,Z 53.878,A 180.000,B 0.000,C 180.000} C_DIS
LIN {X 35.460,Y 29.076,Z 53.873,A 180.000,B 0.000,C 180.000} C_DIS
LIN {X 35.616,Y 29.055,Z 53.869,A 180.000,B 0.000,C 180.000} C_DIS
LIN {X 35.773,Y 29.040,Z 53.864,A 180.000,B 0.000,C 180.000} C_DIS
LIN {X 35.930,Y 29.025,Z 53.859,A 180.000,B 0.000,C 180.000} C_DIS
LIN {X 36.087,Y 29.014,Z 53.854,A 180.000,B 0.000,C 180.000} C_DIS
LIN {X 36.166,Y 29.012,Z 53.851,A 180.000,B 0.000,C 180.000} C_DIS
LIN {X 36.244,Y 29.009,Z 53.849,A 180.000,B 0.000,C 180.000} C_DIS
LIN {X 36.323,Y 29.007,Z 53.846,A 180.000,B 0.000,C 180.000} C_DIS
LIN {X 36.481,Y 29.002,Z 53.841,A 180.000,B 0.000,C 180.000} C_DIS
LIN {X 36.559,Y 29.003,Z 53.839,A 180.000,B 0.000,C 180.000} C_DIS
LIN {X 36.638,Y 29.006,Z 53.836,A 180.000,B 0.000,C 180.000} C_DIS
LIN {X 36.796,Y 29.011,Z 53.831,A 180.000,B 0.000,C 180.000} C_DIS
LIN {X 36.953,Y 29.015,Z 53.825,A 180.000,B 0.000,C 180.000} C_DIS
LIN {X 37.031,Y 29.022,Z 53.823,A 180.000,B 0.000,C 180.000} C_DIS
LIN {X 37.188,Y 29.037,Z 53.817,A 180.000,B 0.000,C 180.000} C_DIS
LIN {X 37.345,Y 29.051,Z 53.812,A 180.000,B 0.000,C 180.000} C_DIS
LIN {X 37.423,Y 29.059,Z 53.809,A 180.000,B 0.000,C 180.000} C_DIS
LIN {X 37.501,Y 29.070,Z 53.806,A 180.000,B 0.000,C 180.000} C_DIS
LIN {X 37.657,Y 29.095,Z 53.801,A 180.000,B 0.000,C 180.000} C_DIS
LIN {X 37.890,Y 29.132,Z 53.793,A 180.000,B 0.000,C 180.000} C_DIS
LIN {X 37.967,Y 29.148,Z 53.790,A 180.000,B 0.000,C 180.000} C_DIS
LIN {X 38.198,Y 29.200,Z 53.782,A 180.000,B 0.000,C 180.000} C_DIS
LIN {X 38.352,Y 29.234,Z 53.776,A 180.000,B 0.000,C 180.000} C_DIS
LIN {X 38.428,Y 29.255,Z 53.774,A 180.000,B 0.000,C 180.000} C_DIS
LIN {X 38.579,Y 29.299,Z 53.768,A 180.000,B 0.000,C 180.000} C_DIS
LIN {X 38.806,Y 29.365,Z 53.760,A 180.000,B 0.000,C 180.000} C_DIS
LIN {X 38.880,Y 29.391,Z 53.757,A 180.000,B 0.000,C 180.000} C_DIS
LIN {X 39.102,Y 29.471,Z 53.749,A 180.000,B 0.000,C 180.000} C_DIS
LIN {X 39.251,Y 29.524,Z 53.743,A 180.000,B 0.000,C 180.000} C_DIS
LIN {X 39.323,Y 29.555,Z 53.741,A 180.000,B 0.000,C 180.000} C_DIS
LIN {X 39.468,Y 29.617,Z 53.735,A 180.000,B 0.000,C 180.000} C_DIS
LIN {X 39.684,Y 29.711,Z 53.727,A 180.000,B 0.000,C 180.000} C_DIS
LIN {X 39.755,Y 29.747,Z 53.724,A 180.000,B 0.000,C 180.000} C_DIS
LIN {X 40.036,Y 29.890,Z 53.713,A 180.000,B 0.000,C 180.000} C_DIS
LIN {X 40.106,Y 29.925,Z 53.710,A 180.000,B 0.000,C 180.000} C_DIS
LIN {X 40.174,Y 29.965,Z 53.708,A 180.000,B 0.000,C 180.000} C_DIS
LIN {X 40.309,Y 30.045,Z 53.702,A 180.000,B 0.000,C 180.000} C_DIS
LIN {X 40.513,Y 30.165,Z 53.694,A 180.000,B 0.000,C 180.000} C_DIS
LIN {X 40.578,Y 30.209,Z 53.691,A 180.000,B 0.000,C 180.000} C_DIS
LIN {X 40.904,Y 30.431,Z 53.677,A 180.000,B 0.000,C 180.000} C_DIS
LIN {X 40.966,Y 30.479,Z 53.675,A 180.000,B 0.000,C 180.000} C_DIS
LIN {X 41.091,Y 30.575,Z 53.669,A 180.000,B 0.000,C 180.000} C_DIS
LIN {X 41.277,Y 30.720,Z 53.661,A 180.000,B 0.000,C 180.000} C_DIS
LIN {X 41.337,Y 30.772,Z 53.658,A 180.000,B 0.000,C 180.000} C_DIS
LIN {X 41.632,Y 31.033,Z 53.644,A 180.000,B 0.000,C 180.000} C_DIS
LIN {X 41.688,Y 31.088,Z 53.642,A 180.000,B 0.000,C 180.000} C_DIS
LIN {X 41.855,Y 31.255,Z 53.633,A 180.000,B 0.000,C 180.000} C_DIS
LIN {X 41.966,Y 31.367,Z 53.628,A 180.000,B 0.000,C 180.000} C_DIS
LIN {X 42.070,Y 31.485,Z 53.622,A 180.000,B 0.000,C 180.000} C_DIS
LIN {X 42.175,Y 31.603,Z 53.617,A 180.000,B 0.000,C 180.000} C_DIS
LIN {X 42.227,Y 31.662,Z 53.614,A 180.000,B 0.000,C 180.000} C_DIS
LIN {X 42.279,Y 31.721,Z 53.611,A 180.000,B 0.000,C 180.000} C_DIS
LIN {X 42.520,Y 32.032,Z 53.598,A 180.000,B 0.000,C 180.000} C_DIS
LIN {X 42.568,Y 32.095,Z 53.595,A 180.000,B 0.000,C 180.000} C_DIS
LIN {X 42.790,Y 32.420,Z 53.581,A 180.000,B 0.000,C 180.000} C_DIS
LIN {X 42.834,Y 32.486,Z 53.578,A 180.000,B 0.000,C 180.000} C_DIS
LIN {X 43.034,Y 32.825,Z 53.565,A 180.000,B 0.000,C 180.000} C_DIS
LIN {X 43.074,Y 32.893,Z 53.562,A 180.000,B 0.000,C 180.000} C_DIS
LIN {X 43.253,Y 33.243,Z 53.548,A 180.000,B 0.000,C 180.000} C_DIS
LIN {X 43.288,Y 33.314,Z 53.545,A 180.000,B 0.000,C 180.000} C_DIS
LIN {X 43.444,Y 33.675,Z 53.532,A 180.000,B 0.000,C 180.000} C_DIS
LIN {X 43.475,Y 33.748,Z 53.529,A 180.000,B 0.000,C 180.000} C_DIS
LIN {X 43.608,Y 34.118,Z 53.515,A 180.000,B 0.000,C 180.000} C_DIS
LIN {X 43.635,Y 34.192,Z 53.512,A 180.000,B 0.000,C 180.000} C_DIS
LIN {X 43.744,Y 34.571,Z 53.499,A 180.000,B 0.000,C 180.000} C_DIS
LIN {X 43.766,Y 34.646,Z 53.496,A 180.000,B 0.000,C 180.000} C_DIS
LIN {X 43.852,Y 35.031,Z 53.482,A 180.000,B 0.000,C 180.000} C_DIS
LIN {X 43.868,Y 35.108,Z 53.479,A 180.000,B 0.000,C 180.000} C_DIS
LIN {X 43.930,Y 35.497,Z 53.466,A 180.000,B 0.000,C 180.000} C_DIS
LIN {X 43.941,Y 35.575,Z 53.463,A 180.000,B 0.000,C 180.000} C_DIS
LIN {X 43.978,Y 35.967,Z 53.449,A 180.000,B 0.000,C 180.000} C_DIS
LIN {X 43.984,Y 36.045,Z 53.446,A 180.000,B 0.000,C 180.000} C_DIS
LIN {X 43.997,Y 36.439,Z 53.433,A 180.000,B 0.000,C 180.000} C_DIS
LIN {X 43.998,Y 36.518,Z 53.430,A 180.000,B 0.000,C 180.000} C_DIS
LIN {X 43.986,Y 36.911,Z 53.416,A 180.000,B 0.000,C 180.000} C_DIS
LIN {X 43.982,Y 36.990,Z 53.413,A 180.000,B 0.000,C 180.000} C_DIS
LIN {X 43.960,Y 37.225,Z 53.405,A 180.000,B 0.000,C 180.000} C_DIS
LIN {X 43.945,Y 37.382,Z 53.400,A 180.000,B 0.000,C 180.000} C_DIS
LIN {X 43.936,Y 37.460,Z 53.397,A 180.000,B 0.000,C 180.000} C_DIS
LIN {X 43.875,Y 37.849,Z 53.383,A 180.000,B 0.000,C 180.000} C_DIS
LIN {X 43.861,Y 37.926,Z 53.380,A 180.000,B 0.000,C 180.000} C_DIS
LIN {X 43.827,Y 38.080,Z 53.375,A 180.000,B 0.000,C 180.000} C_DIS
LIN {X 43.775,Y 38.311,Z 53.367,A 180.000,B 0.000,C 180.000} C_DIS
LIN {X 43.757,Y 38.387,Z 53.364,A 180.000,B 0.000,C 180.000} C_DIS
LIN {X 43.647,Y 38.765,Z 53.350,A 180.000,B 0.000,C 180.000} C_DIS
LIN {X 43.623,Y 38.841,Z 53.347,A 180.000,B 0.000,C 180.000} C_DIS
LIN {X 43.597,Y 38.915,Z 53.345,A 180.000,B 0.000,C 180.000} C_DIS
LIN {X 43.517,Y 39.137,Z 53.336,A 180.000,B 0.000,C 180.000} C_DIS
LIN {X 43.490,Y 39.211,Z 53.334,A 180.000,B 0.000,C 180.000} C_DIS
LIN {X 43.462,Y 39.285,Z 53.331,A 180.000,B 0.000,C 180.000} C_DIS
LIN {X 43.305,Y 39.646,Z 53.317,A 180.000,B 0.000,C 180.000} C_DIS
LIN {X 43.272,Y 39.718,Z 53.314,A 180.000,B 0.000,C 180.000} C_DIS
LIN {X 43.237,Y 39.788,Z 53.312,A 180.000,B 0.000,C 180.000} C_DIS
LIN {X 43.165,Y 39.928,Z 53.306,A 180.000,B 0.000,C 180.000} C_DIS
LIN {X 43.094,Y 40.068,Z 53.301,A 180.000,B 0.000,C 180.000} C_DIS
LIN {X 43.056,Y 40.138,Z 53.298,A 180.000,B 0.000,C 180.000} C_DIS
LIN {X 42.976,Y 40.273,Z 53.292,A 180.000,B 0.000,C 180.000} C_DIS
LIN {X 42.936,Y 40.341,Z 53.290,A 180.000,B 0.000,C 180.000} C_DIS
LIN {X 42.856,Y 40.477,Z 53.284,A 180.000,B 0.000,C 180.000} C_DIS
LIN {X 42.814,Y 40.543,Z 53.281,A 180.000,B 0.000,C 180.000} C_DIS
LIN {X 42.770,Y 40.609,Z 53.279,A 180.000,B 0.000,C 180.000} C_DIS
LIN {X 42.681,Y 40.739,Z 53.273,A 180.000,B 0.000,C 180.000} C_DIS
LIN {X 42.593,Y 40.869,Z 53.268,A 180.000,B 0.000,C 180.000} C_DIS
LIN {X 42.547,Y 40.933,Z 53.265,A 180.000,B 0.000,C 180.000} C_DIS
LIN {X 42.450,Y 41.058,Z 53.259,A 180.000,B 0.000,C 180.000} C_DIS
LIN {X 42.402,Y 41.120,Z 53.257,A 180.000,B 0.000,C 180.000} C_DIS
LIN {X 42.306,Y 41.244,Z 53.251,A 180.000,B 0.000,C 180.000} C_DIS
LIN {X 42.256,Y 41.305,Z 53.248,A 180.000,B 0.000,C 180.000} C_DIS
LIN {X 42.204,Y 41.364,Z 53.246,A 180.000,B 0.000,C 180.000} C_DIS
LIN {X 42.099,Y 41.482,Z 53.240,A 180.000,B 0.000,C 180.000} C_DIS
LIN {X 41.995,Y 41.601,Z 53.235,A 180.000,B 0.000,C 180.000} C_DIS
LIN {X 41.942,Y 41.658,Z 53.232,A 180.000,B 0.000,C 180.000} C_DIS
LIN {X 41.830,Y 41.769,Z 53.226,A 180.000,B 0.000,C 180.000} C_DIS
LIN {X 41.774,Y 41.825,Z 53.224,A 180.000,B 0.000,C 180.000} C_DIS
LIN {X 41.663,Y 41.937,Z 53.218,A 180.000,B 0.000,C 180.000} C_DIS
LIN {X 41.606,Y 41.991,Z 53.215,A 180.000,B 0.000,C 180.000} C_DIS
LIN {X 41.547,Y 42.043,Z 53.213,A 180.000,B 0.000,C 180.000} C_DIS
LIN {X 41.429,Y 42.147,Z 53.207,A 180.000,B 0.000,C 180.000} C_DIS
LIN {X 41.310,Y 42.251,Z 53.202,A 180.000,B 0.000,C 180.000} C_DIS
LIN {X 41.250,Y 42.301,Z 53.199,A 180.000,B 0.000,C 180.000} C_DIS
LIN {X 41.125,Y 42.398,Z 53.193,A 180.000,B 0.000,C 180.000} C_DIS
LIN {X 40.939,Y 42.543,Z 53.185,A 180.000,B 0.000,C 180.000} C_DIS
LIN {X 40.875,Y 42.589,Z 53.182,A 180.000,B 0.000,C 180.000} C_DIS
LIN {X 40.745,Y 42.677,Z 53.177,A 180.000,B 0.000,C 180.000} C_DIS
LIN {X 40.614,Y 42.766,Z 53.172,A 180.000,B 0.000,C 180.000} C_DIS
LIN {X 40.549,Y 42.810,Z 53.169,A 180.000,B 0.000,C 180.000} C_DIS
LIN {X 40.483,Y 42.852,Z 53.166,A 180.000,B 0.000,C 180.000} C_DIS
LIN {X 40.347,Y 42.932,Z 53.161,A 180.000,B 0.000,C 180.000} C_DIS
LIN {X 40.279,Y 42.973,Z 53.159,A 180.000,B 0.000,C 180.000} C_DIS
LIN {X 40.212,Y 43.013,Z 53.156,A 180.000,B 0.000,C 180.000} C_DIS
LIN {X 40.144,Y 43.053,Z 53.154,A 180.000,B 0.000,C 180.000} C_DIS
LIN {X 40.075,Y 43.090,Z 53.151,A 180.000,B 0.000,C 180.000} C_DIS
LIN {X 40.005,Y 43.126,Z 53.149,A 180.000,B 0.000,C 180.000} C_DIS
LIN {X 39.864,Y 43.198,Z 53.144,A 180.000,B 0.000,C 180.000} C_DIS
LIN {X 39.724,Y 43.269,Z 53.139,A 180.000,B 0.000,C 180.000} C_DIS
LIN {X 39.580,Y 43.334,Z 53.134,A 180.000,B 0.000,C 180.000} C_DIS
LIN {X 39.436,Y 43.396,Z 53.129,A 180.000,B 0.000,C 180.000} C_DIS
LIN {X 39.291,Y 43.459,Z 53.124,A 180.000,B 0.000,C 180.000} C_DIS
LIN {X 39.144,Y 43.514,Z 53.120,A 180.000,B 0.000,C 180.000} C_DIS
LIN {X 38.995,Y 43.568,Z 53.115,A 180.000,B 0.000,C 180.000} C_DIS
LIN {X 38.847,Y 43.621,Z 53.111,A 180.000,B 0.000,C 180.000} C_DIS
LIN {X 38.697,Y 43.667,Z 53.106,A 180.000,B 0.000,C 180.000} C_DIS
LIN {X 38.545,Y 43.711,Z 53.102,A 180.000,B 0.000,C 180.000} C_DIS
LIN {X 38.394,Y 43.755,Z 53.097,A 180.000,B 0.000,C 180.000} C_DIS
LIN {X 38.241,Y 43.791,Z 53.093,A 180.000,B 0.000,C 180.000} C_DIS
LIN {X 38.087,Y 43.825,Z 53.089,A 180.000,B 0.000,C 180.000} C_DIS
LIN {X 37.933,Y 43.860,Z 53.085,A 180.000,B 0.000,C 180.000} C_DIS
LIN {X 37.778,Y 43.886,Z 53.081,A 180.000,B 0.000,C 180.000} C_DIS
LIN {X 37.623,Y 43.911,Z 53.077,A 180.000,B 0.000,C 180.000} C_DIS
LIN {X 37.467,Y 43.935,Z 53.073,A 180.000,B 0.000,C 180.000} C_DIS
LIN {X 37.310,Y 43.952,Z 53.070,A 180.000,B 0.000,C 180.000} C_DIS
LIN {X 37.154,Y 43.967,Z 53.066,A 180.000,B 0.000,C 180.000} C_DIS
LIN {X 36.997,Y 43.982,Z 53.062,A 180.000,B 0.000,C 180.000} C_DIS
LIN {X 36.839,Y 43.988,Z 53.059,A 180.000,B 0.000,C 180.000} C_DIS
LIN {X 36.682,Y 43.993,Z 53.056,A 180.000,B 0.000,C 180.000} C_DIS
LIN {X 36.525,Y 43.998,Z 53.052,A 180.000,B 0.000,C 180.000} C_DIS
LIN {X 36.367,Y 43.995,Z 53.049,A 180.000,B 0.000,C 180.000} C_DIS
LIN {X 36.210,Y 43.990,Z 53.046,A 180.000,B 0.000,C 180.000} C_DIS
LIN {X 36.052,Y 43.985,Z 53.043,A 180.000,B 0.000,C 180.000} C_DIS
LIN {X 35.895,Y 43.971,Z 53.040,A 180.000,B 0.000,C 180.000} C_DIS
LIN {X 35.739,Y 43.957,Z 53.037,A 180.000,B 0.000,C 180.000} C_DIS
LIN {X 35.582,Y 43.942,Z 53.034,A 180.000,B 0.000,C 180.000} C_DIS
LIN {X 35.426,Y 43.918,Z 53.032,A 180.000,B 0.000,C 180.000} C_DIS
LIN {X 35.270,Y 43.894,Z 53.029,A 180.000,B 0.000,C 180.000} C_DIS
LIN {X 35.115,Y 43.869,Z 53.027,A 180.000,B 0.000,C 180.000} C_DIS
LIN {X 34.807,Y 43.802,Z 53.022,A 180.000,B 0.000,C 180.000} C_DIS
LIN {X 34.502,Y 43.724,Z 53.018,A 180.000,B 0.000,C 180.000} C_DIS
LIN {X 34.199,Y 43.637,Z 53.014,A 180.000,B 0.000,C 180.000} C_DIS
LIN {X 33.903,Y 43.531,Z 53.011,A 180.000,B 0.000,C 180.000} C_DIS
LIN {X 33.609,Y 43.416,Z 53.008,A 180.000,B 0.000,C 180.000} C_DIS
LIN {X 33.320,Y 43.291,Z 53.005,A 180.000,B 0.000,C 180.000} C_DIS
LIN {X 33.039,Y 43.149,Z 53.003,A 180.000,B 0.000,C 180.000} C_DIS
LIN {X 32.763,Y 42.998,Z 53.002,A 180.000,B 0.000,C 180.000} C_DIS
LIN {X 32.492,Y 42.837,Z 53.001,A 180.000,B 0.000,C 180.000} C_DIS
LIN {X 32.231,Y 42.661,Z 53.000,A 180.000,B 0.000,C 180.000} C_DIS
LIN {X 32.040,Y 42.526,Z 53.000,A 180.000,B 0.000,C 180.000} C_DIS
; Cutting Move Starts
LIN {X 31.824,Y 42.359,Z 53.000,A 180.000,B 0.000,C 180.000} C_DIS
LIN {X 31.646,Y 42.212,Z 53.000,A 180.000,B 0.000,C 180.000} C_DIS
LIN {X 31.421,Y 42.014,Z 53.000,A 180.000,B 0.000,C 180.000} C_DIS
LIN {X 31.288,Y 41.888,Z 53.000,A 180.000,B 0.000,C 180.000} C_DIS
LIN {X 31.057,Y 41.657,Z 53.000,A 180.000,B 0.000,C 180.000} C_DIS
LIN {X 30.930,Y 41.516,Z 53.000,A 180.000,B 0.000,C 180.000} C_DIS
LIN {X 30.739,Y 41.299,Z 53.000,A 180.000,B 0.000,C 180.000} C_DIS
LIN {X 30.598,Y 41.120,Z 53.000,A 180.000,B 0.000,C 180.000} C_DIS
LIN {X 30.460,Y 40.942,Z 53.000,A 180.000,B 0.000,C 180.000} C_DIS
LIN {X 30.394,Y 40.850,Z 53.000,A 180.000,B 0.000,C 180.000} C_DIS
LIN {X 30.213,Y 40.584,Z 53.000,A 180.000,B 0.000,C 180.000} C_DIS
LIN {X 30.102,Y 40.405,Z 53.000,A 180.000,B 0.000,C 180.000} C_DIS
LIN {X 29.996,Y 40.226,Z 53.000,A 180.000,B 0.000,C 180.000} C_DIS
LIN {X 29.896,Y 40.048,Z 53.000,A 180.000,B 0.000,C 180.000} C_DIS
LIN {X 29.805,Y 39.869,Z 53.000,A 180.000,B 0.000,C 180.000} C_DIS
LIN {X 29.714,Y 39.690,Z 53.000,A 180.000,B 0.000,C 180.000} C_DIS
LIN {X 29.559,Y 39.333,Z 53.000,A 180.000,B 0.000,C 180.000} C_DIS
LIN {X 29.500,Y 39.184,Z 53.000,A 180.000,B 0.000,C 180.000} C_DIS
LIN {X 29.425,Y 38.975,Z 53.000,A 180.000,B 0.000,C 180.000} C_DIS
LIN {X 29.362,Y 38.796,Z 53.000,A 180.000,B 0.000,C 180.000} C_DIS
LIN {X 29.258,Y 38.439,Z 53.000,A 180.000,B 0.000,C 180.000} C_DIS
LIN {X 29.213,Y 38.260,Z 53.000,A 180.000,B 0.000,C 180.000} C_DIS
LIN {X 29.143,Y 37.944,Z 53.000,A 180.000,B 0.000,C 180.000} C_DIS
LIN {X 29.134,Y 37.902,Z 53.000,A 180.000,B 0.000,C 180.000} C_DIS
LIN {X 29.077,Y 37.545,Z 53.000,A 180.000,B 0.000,C 180.000} C_DIS
LIN {X 29.053,Y 37.366,Z 53.000,A 180.000,B 0.000,C 180.000} C_DIS
LIN {X 29.020,Y 37.009,Z 53.000,A 180.000,B 0.000,C 180.000} C_DIS
LIN {X 29.012,Y 36.830,Z 53.000,A 180.000,B 0.000,C 180.000} C_DIS
LIN {X 29.006,Y 36.651,Z 53.000,A 180.000,B 0.000,C 180.000} C_DIS
LIN {X 29.002,Y 36.472,Z 53.000,A 180.000,B 0.000,C 180.000} C_DIS
LIN {X 29.013,Y 36.115,Z 53.000,A 180.000,B 0.000,C 180.000} C_DIS
LIN {X 29.025,Y 35.936,Z 53.000,A 180.000,B 0.000,C 180.000} C_DIS
LIN {X 29.059,Y 35.578,Z 53.000,A 180.000,B 0.000,C 180.000} C_DIS
LIN {X 29.086,Y 35.400,Z 53.000,A 180.000,B 0.000,C 180.000} C_DIS
LIN {X 29.114,Y 35.221,Z 53.000,A 180.000,B 0.000,C 180.000} C_DIS
LIN {X 29.143,Y 35.056,Z 53.000,A 180.000,B 0.000,C 180.000} C_DIS
LIN {X 29.226,Y 34.685,Z 53.000,A 180.000,B 0.000,C 180.000} C_DIS
LIN {X 29.274,Y 34.506,Z 53.000,A 180.000,B 0.000,C 180.000} C_DIS
LIN {X 29.326,Y 34.327,Z 53.000,A 180.000,B 0.000,C 180.000} C_DIS
LIN {X 29.381,Y 34.148,Z 53.000,A 180.000,B 0.000,C 180.000} C_DIS
LIN {X 29.509,Y 33.791,Z 53.000,A 180.000,B 0.000,C 180.000} C_DIS
LIN {X 29.583,Y 33.612,Z 53.000,A 180.000,B 0.000,C 180.000} C_DIS
LIN {X 29.679,Y 33.390,Z 53.000,A 180.000,B 0.000,C 180.000} C_DIS
LIN {X 29.742,Y 33.254,Z 53.000,A 180.000,B 0.000,C 180.000} C_DIS
LIN {X 29.924,Y 32.897,Z 53.000,A 180.000,B 0.000,C 180.000} C_DIS
LIN {X 30.029,Y 32.718,Z 53.000,A 180.000,B 0.000,C 180.000} C_DIS
LIN {X 30.135,Y 32.539,Z 53.000,A 180.000,B 0.000,C 180.000} C_DIS
LIN {X 30.215,Y 32.413,Z 53.000,A 180.000,B 0.000,C 180.000} C_DIS
LIN {X 30.394,Y 32.150,Z 53.000,A 180.000,B 0.000,C 180.000} C_DIS
LIN {X 30.503,Y 32.003,Z 53.000,A 180.000,B 0.000,C 180.000} C_DIS
LIN {X 30.641,Y 31.824,Z 53.000,A 180.000,B 0.000,C 180.000} C_DIS
LIN {X 30.752,Y 31.687,Z 53.000,A 180.000,B 0.000,C 180.000} C_DIS
LIN {X 30.945,Y 31.467,Z 53.000,A 180.000,B 0.000,C 180.000} C_DIS
LIN {X 31.109,Y 31.291,Z 53.000,A 180.000,B 0.000,C 180.000} C_DIS
LIN {X 31.291,Y 31.109,Z 53.000,A 180.000,B 0.000,C 180.000} C_DIS
LIN {X 31.467,Y 30.945,Z 53.000,A 180.000,B 0.000,C 180.000} C_DIS
LIN {X 31.687,Y 30.752,Z 53.000,A 180.000,B 0.000,C 180.000} C_DIS
LIN {X 31.824,Y 30.641,Z 53.000,A 180.000,B 0.000,C 180.000} C_DIS
LIN {X 32.003,Y 30.503,Z 53.000,A 180.000,B 0.000,C 180.000} C_DIS
LIN {X 32.150,Y 30.394,Z 53.000,A 180.000,B 0.000,C 180.000} C_DIS
LIN {X 32.413,Y 30.215,Z 53.000,A 180.000,B 0.000,C 180.000} C_DIS
LIN {X 32.539,Y 30.135,Z 53.000,A 180.000,B 0.000,C 180.000} C_DIS
LIN {X 32.718,Y 30.029,Z 53.000,A 180.000,B 0.000,C 180.000} C_DIS
LIN {X 32.897,Y 29.924,Z 53.000,A 180.000,B 0.000,C 180.000} C_DIS
LIN {X 33.254,Y 29.742,Z 53.000,A 180.000,B 0.000,C 180.000} C_DIS
LIN {X 33.390,Y 29.679,Z 53.000,A 180.000,B 0.000,C 180.000} C_DIS
LIN {X 33.612,Y 29.583,Z 53.000,A 180.000,B 0.000,C 180.000} C_DIS
LIN {X 33.791,Y 29.509,Z 53.000,A 180.000,B 0.000,C 180.000} C_DIS
LIN {X 34.148,Y 29.381,Z 53.000,A 180.000,B 0.000,C 180.000} C_DIS
LIN {X 34.327,Y 29.326,Z 53.000,A 180.000,B 0.000,C 180.000} C_DIS
LIN {X 34.506,Y 29.274,Z 53.000,A 180.000,B 0.000,C 180.000} C_DIS
LIN {X 34.685,Y 29.226,Z 53.000,A 180.000,B 0.000,C 180.000} C_DIS
LIN {X 35.056,Y 29.143,Z 53.000,A 180.000,B 0.000,C 180.000} C_DIS
LIN {X 35.221,Y 29.114,Z 53.000,A 180.000,B 0.000,C 180.000} C_DIS
LIN {X 35.400,Y 29.086,Z 53.000,A 180.000,B 0.000,C 180.000} C_DIS
LIN {X 35.578,Y 29.059,Z 53.000,A 180.000,B 0.000,C 180.000} C_DIS
LIN {X 35.936,Y 29.025,Z 53.000,A 180.000,B 0.000,C 180.000} C_DIS
LIN {X 36.115,Y 29.013,Z 53.000,A 180.000,B 0.000,C 180.000} C_DIS
LIN {X 36.472,Y 29.002,Z 53.000,A 180.000,B 0.000,C 180.000} C_DIS
LIN {X 36.651,Y 29.006,Z 53.000,A 180.000,B 0.000,C 180.000} C_DIS
LIN {X 36.830,Y 29.012,Z 53.000,A 180.000,B 0.000,C 180.000} C_DIS
LIN {X 37.009,Y 29.020,Z 53.000,A 180.000,B 0.000,C 180.000} C_DIS
LIN {X 37.366,Y 29.053,Z 53.000,A 180.000,B 0.000,C 180.000} C_DIS
LIN {X 37.545,Y 29.077,Z 53.000,A 180.000,B 0.000,C 180.000} C_DIS
LIN {X 37.902,Y 29.134,Z 53.000,A 180.000,B 0.000,C 180.000} C_DIS
LIN {X 37.944,Y 29.143,Z 53.000,A 180.000,B 0.000,C 180.000} C_DIS
LIN {X 38.260,Y 29.213,Z 53.000,A 180.000,B 0.000,C 180.000} C_DIS
LIN {X 38.439,Y 29.258,Z 53.000,A 180.000,B 0.000,C 180.000} C_DIS
LIN {X 38.796,Y 29.362,Z 53.000,A 180.000,B 0.000,C 180.000} C_DIS
LIN {X 38.975,Y 29.425,Z 53.000,A 180.000,B 0.000,C 180.000} C_DIS
LIN {X 39.184,Y 29.500,Z 53.000,A 180.000,B 0.000,C 180.000} C_DIS
LIN {X 39.333,Y 29.559,Z 53.000,A 180.000,B 0.000,C 180.000} C_DIS
LIN {X 39.690,Y 29.714,Z 53.000,A 180.000,B 0.000,C 180.000} C_DIS
LIN {X 39.869,Y 29.805,Z 53.000,A 180.000,B 0.000,C 180.000} C_DIS
LIN {X 40.048,Y 29.896,Z 53.000,A 180.000,B 0.000,C 180.000} C_DIS
LIN {X 40.226,Y 29.996,Z 53.000,A 180.000,B 0.000,C 180.000} C_DIS
LIN {X 40.405,Y 30.102,Z 53.000,A 180.000,B 0.000,C 180.000} C_DIS
LIN {X 40.584,Y 30.213,Z 53.000,A 180.000,B 0.000,C 180.000} C_DIS
LIN {X 40.850,Y 30.394,Z 53.000,A 180.000,B 0.000,C 180.000} C_DIS
LIN {X 40.942,Y 30.460,Z 53.000,A 180.000,B 0.000,C 180.000} C_DIS
LIN {X 41.120,Y 30.598,Z 53.000,A 180.000,B 0.000,C 180.000} C_DIS
LIN {X 41.299,Y 30.739,Z 53.000,A 180.000,B 0.000,C 180.000} C_DIS
LIN {X 41.516,Y 30.930,Z 53.000,A 180.000,B 0.000,C 180.000} C_DIS
LIN {X 41.657,Y 31.057,Z 53.000,A 180.000,B 0.000,C 180.000} C_DIS
LIN {X 41.888,Y 31.288,Z 53.000,A 180.000,B 0.000,C 180.000} C_DIS
LIN {X 42.014,Y 31.421,Z 53.000,A 180.000,B 0.000,C 180.000} C_DIS
LIN {X 42.212,Y 31.646,Z 53.000,A 180.000,B 0.000,C 180.000} C_DIS
LIN {X 42.359,Y 31.824,Z 53.000,A 180.000,B 0.000,C 180.000} C_DIS
LIN {X 42.550,Y 32.072,Z 53.000,A 180.000,B 0.000,C 180.000} C_DIS
LIN {X 42.627,Y 32.182,Z 53.000,A 180.000,B 0.000,C 180.000} C_DIS
LIN {X 42.749,Y 32.361,Z 53.000,A 180.000,B 0.000,C 180.000} C_DIS
LIN {X 42.865,Y 32.539,Z 53.000,A 180.000,B 0.000,C 180.000} C_DIS
LIN {X 42.971,Y 32.718,Z 53.000,A 180.000,B 0.000,C 180.000} C_DIS
LIN {X 43.076,Y 32.897,Z 53.000,A 180.000,B 0.000,C 180.000} C_DIS
LIN {X 43.266,Y 33.269,Z 53.000,A 180.000,B 0.000,C 180.000} C_DIS
LIN {X 43.340,Y 33.433,Z 53.000,A 180.000,B 0.000,C 180.000} C_DIS
LIN {X 43.444,Y 33.675,Z 53.000,A 180.000,B 0.000,C 180.000} C_DIS
LIN {X 43.491,Y 33.791,Z 53.000,A 180.000,B 0.000,C 180.000} C_DIS
LIN {X 43.623,Y 34.159,Z 53.000,A 180.000,B 0.000,C 180.000} C_DIS
LIN {X 43.674,Y 34.327,Z 53.000,A 180.000,B 0.000,C 180.000} C_DIS
LIN {X 43.726,Y 34.506,Z 53.000,A 180.000,B 0.000,C 180.000} C_DIS
LIN {X 43.774,Y 34.685,Z 53.000,A 180.000,B 0.000,C 180.000} C_DIS
LIN {X 43.854,Y 35.042,Z 53.000,A 180.000,B 0.000,C 180.000} C_DIS
LIN {X 43.886,Y 35.221,Z 53.000,A 180.000,B 0.000,C 180.000} C_DIS
LIN {X 43.914,Y 35.400,Z 53.000,A 180.000,B 0.000,C 180.000} C_DIS
LIN {X 43.941,Y 35.578,Z 53.000,A 180.000,B 0.000,C 180.000} C_DIS
LIN {X 43.981,Y 35.994,Z 53.000,A 180.000,B 0.000,C 180.000} C_DIS
LIN {X 43.987,Y 36.115,Z 53.000,A 180.000,B 0.000,C 180.000} C_DIS
LIN {X 43.998,Y 36.472,Z 53.000,A 180.000,B 0.000,C 180.000} C_DIS
LIN {X 43.994,Y 36.651,Z 53.000,A 180.000,B 0.000,C 180.000} C_DIS
LIN {X 43.988,Y 36.830,Z 53.000,A 180.000,B 0.000,C 180.000} C_DIS
LIN {X 43.981,Y 37.006,Z 53.000,A 180.000,B 0.000,C 180.000} C_DIS
LIN {X 43.947,Y 37.366,Z 53.000,A 180.000,B 0.000,C 180.000} C_DIS
LIN {X 43.923,Y 37.545,Z 53.000,A 180.000,B 0.000,C 180.000} C_DIS
LIN {X 43.866,Y 37.902,Z 53.000,A 180.000,B 0.000,C 180.000} C_DIS
LIN {X 43.827,Y 38.081,Z 53.000,A 180.000,B 0.000,C 180.000} C_DIS
LIN {X 43.787,Y 38.260,Z 53.000,A 180.000,B 0.000,C 180.000} C_DIS
LIN {X 43.742,Y 38.439,Z 53.000,A 180.000,B 0.000,C 180.000} C_DIS
LIN {X 43.638,Y 38.796,Z 53.000,A 180.000,B 0.000,C 180.000} C_DIS
LIN {X 43.623,Y 38.841,Z 53.000,A 180.000,B 0.000,C 180.000} C_DIS
LIN {X 43.511,Y 39.154,Z 53.000,A 180.000,B 0.000,C 180.000} C_DIS
LIN {X 43.444,Y 39.325,Z 53.000,A 180.000,B 0.000,C 180.000} C_DIS
LIN {X 43.286,Y 39.690,Z 53.000,A 180.000,B 0.000,C 180.000} C_DIS
LIN {X 43.266,Y 39.731,Z 53.000,A 180.000,B 0.000,C 180.000} C_DIS
LIN {X 43.087,Y 40.082,Z 53.000,A 180.000,B 0.000,C 180.000} C_DIS
LIN {X 43.004,Y 40.226,Z 53.000,A 180.000,B 0.000,C 180.000} C_DIS
LIN {X 42.898,Y 40.405,Z 53.000,A 180.000,B 0.000,C 180.000} C_DIS
LIN {X 42.787,Y 40.584,Z 53.000,A 180.000,B 0.000,C 180.000} C_DIS
LIN {X 42.665,Y 40.763,Z 53.000,A 180.000,B 0.000,C 180.000} C_DIS
LIN {X 42.550,Y 40.928,Z 53.000,A 180.000,B 0.000,C 180.000} C_DIS
LIN {X 42.372,Y 41.159,Z 53.000,A 180.000,B 0.000,C 180.000} C_DIS
LIN {X 42.261,Y 41.299,Z 53.000,A 180.000,B 0.000,C 180.000} C_DIS
LIN {X 42.014,Y 41.579,Z 53.000,A 180.000,B 0.000,C 180.000} C_DIS
LIN {X 41.943,Y 41.657,Z 53.000,A 180.000,B 0.000,C 180.000} C_DIS
LIN {X 41.657,Y 41.943,Z 53.000,A 180.000,B 0.000,C 180.000} C_DIS
LIN {X 41.579,Y 42.014,Z 53.000,A 180.000,B 0.000,C 180.000} C_DIS
LIN {X 41.299,Y 42.261,Z 53.000,A 180.000,B 0.000,C 180.000} C_DIS
LIN {X 41.159,Y 42.372,Z 53.000,A 180.000,B 0.000,C 180.000} C_DIS
LIN {X 40.928,Y 42.550,Z 53.000,A 180.000,B 0.000,C 180.000} C_DIS
LIN {X 40.763,Y 42.665,Z 53.000,A 180.000,B 0.000,C 180.000} C_DIS
LIN {X 40.584,Y 42.787,Z 53.000,A 180.000,B 0.000,C 180.000} C_DIS
LIN {X 40.405,Y 42.898,Z 53.000,A 180.000,B 0.000,C 180.000} C_DIS
LIN {X 40.226,Y 43.004,Z 53.000,A 180.000,B 0.000,C 180.000} C_DIS
LIN {X 40.082,Y 43.087,Z 53.000,A 180.000,B 0.000,C 180.000} C_DIS
LIN {X 39.731,Y 43.266,Z 53.000,A 180.000,B 0.000,C 180.000} C_DIS
LIN {X 39.690,Y 43.286,Z 53.000,A 180.000,B 0.000,C 180.000} C_DIS
LIN {X 39.325,Y 43.444,Z 53.000,A 180.000,B 0.000,C 180.000} C_DIS
LIN {X 39.154,Y 43.511,Z 53.000,A 180.000,B 0.000,C 180.000} C_DIS
LIN {X 38.841,Y 43.623,Z 53.000,A 180.000,B 0.000,C 180.000} C_DIS
LIN {X 38.796,Y 43.638,Z 53.000,A 180.000,B 0.000,C 180.000} C_DIS
LIN {X 38.439,Y 43.742,Z 53.000,A 180.000,B 0.000,C 180.000} C_DIS
LIN {X 38.260,Y 43.787,Z 53.000,A 180.000,B 0.000,C 180.000} C_DIS
LIN {X 38.081,Y 43.827,Z 53.000,A 180.000,B 0.000,C 180.000} C_DIS
LIN {X 37.902,Y 43.866,Z 53.000,A 180.000,B 0.000,C 180.000} C_DIS
LIN {X 37.545,Y 43.923,Z 53.000,A 180.000,B 0.000,C 180.000} C_DIS
LIN {X 37.366,Y 43.947,Z 53.000,A 180.000,B 0.000,C 180.000} C_DIS
LIN {X 37.006,Y 43.981,Z 53.000,A 180.000,B 0.000,C 180.000} C_DIS
LIN {X 36.830,Y 43.988,Z 53.000,A 180.000,B 0.000,C 180.000} C_DIS
LIN {X 36.651,Y 43.994,Z 53.000,A 180.000,B 0.000,C 180.000} C_DIS
LIN {X 36.472,Y 43.998,Z 53.000,A 180.000,B 0.000,C 180.000} C_DIS
LIN {X 36.115,Y 43.987,Z 53.000,A 180.000,B 0.000,C 180.000} C_DIS
LIN {X 35.994,Y 43.981,Z 53.000,A 180.000,B 0.000,C 180.000} C_DIS
LIN {X 35.578,Y 43.941,Z 53.000,A 180.000,B 0.000,C 180.000} C_DIS
LIN {X 35.400,Y 43.914,Z 53.000,A 180.000,B 0.000,C 180.000} C_DIS
LIN {X 35.221,Y 43.886,Z 53.000,A 180.000,B 0.000,C 180.000} C_DIS
LIN {X 35.042,Y 43.854,Z 53.000,A 180.000,B 0.000,C 180.000} C_DIS
LIN {X 34.685,Y 43.774,Z 53.000,A 180.000,B 0.000,C 180.000} C_DIS
LIN {X 34.506,Y 43.726,Z 53.000,A 180.000,B 0.000,C 180.000} C_DIS
LIN {X 34.327,Y 43.674,Z 53.000,A 180.000,B 0.000,C 180.000} C_DIS
LIN {X 34.159,Y 43.623,Z 53.000,A 180.000,B 0.000,C 180.000} C_DIS
LIN {X 33.791,Y 43.491,Z 53.000,A 180.000,B 0.000,C 180.000} C_DIS
LIN {X 33.675,Y 43.444,Z 53.000,A 180.000,B 0.000,C 180.000} C_DIS
LIN {X 33.433,Y 43.340,Z 53.000,A 180.000,B 0.000,C 180.000} C_DIS
LIN {X 33.269,Y 43.266,Z 53.000,A 180.000,B 0.000,C 180.000} C_DIS
LIN {X 32.897,Y 43.076,Z 53.000,A 180.000,B 0.000,C 180.000} C_DIS
LIN {X 32.718,Y 42.971,Z 53.000,A 180.000,B 0.000,C 180.000} C_DIS
LIN {X 32.539,Y 42.865,Z 53.000,A 180.000,B 0.000,C 180.000} C_DIS
LIN {X 32.361,Y 42.749,Z 53.000,A 180.000,B 0.000,C 180.000} C_DIS
LIN {X 32.182,Y 42.627,Z 53.000,A 180.000,B 0.000,C 180.000} C_DIS
LIN {X 32.072,Y 42.550,Z 53.000,A 180.000,B 0.000,C 180.000} C_DIS
LIN {X 32.040,Y 42.526,Z 53.000,A 180.000,B 0.000,C 180.000} C_DIS
; Link Move Starts
LIN {X 31.792,Y 42.333,Z 53.000,A 180.000,B 0.000,C 180.000} C_DIS
LIN {X 31.552,Y 42.129,Z 52.999,A 180.000,B 0.000,C 180.000} C_DIS
LIN {X 31.318,Y 41.918,Z 52.998,A 180.000,B 0.000,C 180.000} C_DIS
LIN {X 31.095,Y 41.695,Z 52.996,A 180.000,B 0.000,C 180.000} C_DIS
LIN {X 30.883,Y 41.463,Z 52.994,A 180.000,B 0.000,C 180.000} C_DIS
LIN {X 30.678,Y 41.223,Z 52.991,A 180.000,B 0.000,C 180.000} C_DIS
LIN {X 30.485,Y 40.974,Z 52.988,A 180.000,B 0.000,C 180.000} C_DIS
LIN {X 30.304,Y 40.717,Z 52.985,A 180.000,B 0.000,C 180.000} C_DIS
LIN {X 30.131,Y 40.454,Z 52.981,A 180.000,B 0.000,C 180.000} C_DIS
LIN {X 29.970,Y 40.183,Z 52.977,A 180.000,B 0.000,C 180.000} C_DIS
LIN {X 29.823,Y 39.904,Z 52.972,A 180.000,B 0.000,C 180.000} C_DIS
LIN {X 29.751,Y 39.764,Z 52.969,A 180.000,B 0.000,C 180.000} C_DIS
LIN {X 29.684,Y 39.622,Z 52.967,A 180.000,B 0.000,C 180.000} C_DIS
LIN {X 29.622,Y 39.477,Z 52.964,A 180.000,B 0.000,C 180.000} C_DIS
LIN {X 29.559,Y 39.333,Z 52.961,A 180.000,B 0.000,C 180.000} C_DIS
LIN {X 29.501,Y 39.186,Z 52.959,A 180.000,B 0.000,C 180.000} C_DIS
LIN {X 29.448,Y 39.038,Z 52.956,A 180.000,B 0.000,C 180.000} C_DIS
LIN {X 29.394,Y 38.890,Z 52.952,A 180.000,B 0.000,C 180.000} C_DIS
LIN {X 29.346,Y 38.740,Z 52.949,A 180.000,B 0.000,C 180.000} C_DIS
LIN {X 29.302,Y 38.589,Z 52.946,A 180.000,B 0.000,C 180.000} C_DIS
LIN {X 29.258,Y 38.438,Z 52.943,A 180.000,B 0.000,C 180.000} C_DIS
LIN {X 29.219,Y 38.285,Z 52.939,A 180.000,B 0.000,C 180.000} C_DIS
LIN {X 29.185,Y 38.131,Z 52.936,A 180.000,B 0.000,C 180.000} C_DIS
LIN {X 29.150,Y 37.978,Z 52.932,A 180.000,B 0.000,C 180.000} C_DIS
LIN {X 29.121,Y 37.823,Z 52.928,A 180.000,B 0.000,C 180.000} C_DIS
LIN {X 29.096,Y 37.667,Z 52.925,A 180.000,B 0.000,C 180.000} C_DIS
LIN {X 29.072,Y 37.512,Z 52.921,A 180.000,B 0.000,C 180.000} C_DIS
LIN {X 29.052,Y 37.355,Z 52.917,A 180.000,B 0.000,C 180.000} C_DIS
LIN {X 29.038,Y 37.199,Z 52.913,A 180.000,B 0.000,C 180.000} C_DIS
LIN {X 29.023,Y 37.042,Z 52.909,A 180.000,B 0.000,C 180.000} C_DIS
LIN {X 29.013,Y 36.885,Z 52.905,A 180.000,B 0.000,C 180.000} C_DIS
LIN {X 29.008,Y 36.727,Z 52.900,A 180.000,B 0.000,C 180.000} C_DIS
LIN {X 29.003,Y 36.570,Z 52.896,A 180.000,B 0.000,C 180.000} C_DIS
LIN {X 29.004,Y 36.412,Z 52.892,A 180.000,B 0.000,C 180.000} C_DIS
LIN {X 29.009,Y 36.255,Z 52.887,A 180.000,B 0.000,C 180.000} C_DIS
LIN {X 29.014,Y 36.097,Z 52.883,A 180.000,B 0.000,C 180.000} C_DIS
LIN {X 29.024,Y 35.940,Z 52.878,A 180.000,B 0.000,C 180.000} C_DIS
LIN {X 29.039,Y 35.783,Z 52.873,A 180.000,B 0.000,C 180.000} C_DIS
LIN {X 29.054,Y 35.627,Z 52.869,A 180.000,B 0.000,C 180.000} C_DIS
LIN {X 29.075,Y 35.471,Z 52.864,A 180.000,B 0.000,C 180.000} C_DIS
LIN {X 29.099,Y 35.315,Z 52.859,A 180.000,B 0.000,C 180.000} C_DIS
LIN {X 29.124,Y 35.159,Z 52.854,A 180.000,B 0.000,C 180.000} C_DIS
LIN {X 29.137,Y 35.082,Z 52.851,A 180.000,B 0.000,C 180.000} C_DIS
LIN {X 29.154,Y 35.005,Z 52.849,A 180.000,B 0.000,C 180.000} C_DIS
LIN {X 29.171,Y 34.928,Z 52.846,A 180.000,B 0.000,C 180.000} C_DIS
LIN {X 29.189,Y 34.851,Z 52.844,A 180.000,B 0.000,C 180.000} C_DIS
LIN {X 29.206,Y 34.774,Z 52.841,A 180.000,B 0.000,C 180.000} C_DIS
LIN {X 29.223,Y 34.697,Z 52.839,A 180.000,B 0.000,C 180.000} C_DIS
LIN {X 29.241,Y 34.621,Z 52.836,A 180.000,B 0.000,C 180.000} C_DIS
LIN {X 29.263,Y 34.545,Z 52.833,A 180.000,B 0.000,C 180.000} C_DIS
LIN {X 29.307,Y 34.394,Z 52.828,A 180.000,B 0.000,C 180.000} C_DIS
LIN {X 29.351,Y 34.243,Z 52.823,A 180.000,B 0.000,C 180.000} C_DIS
LIN {X 29.374,Y 34.167,Z 52.820,A 180.000,B 0.000,C 180.000} C_DIS
LIN {X 29.427,Y 34.019,Z 52.815,A 180.000,B 0.000,C 180.000} C_DIS
LIN {X 29.481,Y 33.871,Z 52.809,A 180.000,B 0.000,C 180.000} C_DIS
LIN {X 29.507,Y 33.797,Z 52.806,A 180.000,B 0.000,C 180.000} C_DIS
LIN {X 29.535,Y 33.723,Z 52.804,A 180.000,B 0.000,C 180.000} C_DIS
LIN {X 29.597,Y 33.579,Z 52.798,A 180.000,B 0.000,C 180.000} C_DIS
LIN {X 29.629,Y 33.506,Z 52.796,A 180.000,B 0.000,C 180.000} C_DIS
LIN {X 29.691,Y 33.362,Z 52.790,A 180.000,B 0.000,C 180.000} C_DIS
LIN {X 29.724,Y 33.290,Z 52.787,A 180.000,B 0.000,C 180.000} C_DIS
LIN {X 29.759,Y 33.220,Z 52.785,A 180.000,B 0.000,C 180.000} C_DIS
LIN {X 29.831,Y 33.079,Z 52.779,A 180.000,B 0.000,C 180.000} C_DIS
LIN {X 29.902,Y 32.939,Z 52.774,A 180.000,B 0.000,C 180.000} C_DIS
LIN {X 29.939,Y 32.869,Z 52.771,A 180.000,B 0.000,C 180.000} C_DIS
LIN {X 30.020,Y 32.734,Z 52.765,A 180.000,B 0.000,C 180.000} C_DIS
LIN {X 30.060,Y 32.666,Z 52.763,A 180.000,B 0.000,C 180.000} C_DIS
LIN {X 30.140,Y 32.531,Z 52.757,A 180.000,B 0.000,C 180.000} C_DIS
LIN {X 30.181,Y 32.464,Z 52.754,A 180.000,B 0.000,C 180.000} C_DIS
LIN {X 30.225,Y 32.398,Z 52.752,A 180.000,B 0.000,C 180.000} C_DIS
LIN {X 30.314,Y 32.268,Z 52.746,A 180.000,B 0.000,C 180.000} C_DIS
LIN {X 30.402,Y 32.138,Z 52.741,A 180.000,B 0.000,C 180.000} C_DIS
LIN {X 30.448,Y 32.074,Z 52.738,A 180.000,B 0.000,C 180.000} C_DIS
LIN {X 30.545,Y 31.949,Z 52.732,A 180.000,B 0.000,C 180.000} C_DIS
LIN {X 30.593,Y 31.887,Z 52.730,A 180.000,B 0.000,C 180.000} C_DIS
LIN {X 30.689,Y 31.762,Z 52.724,A 180.000,B 0.000,C 180.000} C_DIS
LIN {X 30.739,Y 31.701,Z 52.721,A 180.000,B 0.000,C 180.000} C_DIS
LIN {X 30.791,Y 31.642,Z 52.719,A 180.000,B 0.000,C 180.000} C_DIS
LIN {X 30.895,Y 31.524,Z 52.713,A 180.000,B 0.000,C 180.000} C_DIS
LIN {X 30.999,Y 31.406,Z 52.708,A 180.000,B 0.000,C 180.000} C_DIS
LIN {X 31.053,Y 31.348,Z 52.705,A 180.000,B 0.000,C 180.000} C_DIS
LIN {X 31.164,Y 31.236,Z 52.699,A 180.000,B 0.000,C 180.000} C_DIS
LIN {X 31.220,Y 31.181,Z 52.697,A 180.000,B 0.000,C 180.000} C_DIS
LIN {X 31.331,Y 31.069,Z 52.691,A 180.000,B 0.000,C 180.000} C_DIS
LIN {X 31.388,Y 31.015,Z 52.688,A 180.000,B 0.000,C 180.000} C_DIS
LIN {X 31.447,Y 30.963,Z 52.686,A 180.000,B 0.000,C 180.000} C_DIS
LIN {X 31.565,Y 30.859,Z 52.680,A 180.000,B 0.000,C 180.000} C_DIS
LIN {X 31.683,Y 30.754,Z 52.675,A 180.000,B 0.000,C 180.000} C_DIS
LIN {X 31.744,Y 30.704,Z 52.672,A 180.000,B 0.000,C 180.000} C_DIS
LIN {X 31.868,Y 30.607,Z 52.666,A 180.000,B 0.000,C 180.000} C_DIS
LIN {X 31.930,Y 30.559,Z 52.664,A 180.000,B 0.000,C 180.000} C_DIS
LIN {X 32.055,Y 30.462,Z 52.658,A 180.000,B 0.000,C 180.000} C_DIS
LIN {X 32.118,Y 30.416,Z 52.655,A 180.000,B 0.000,C 180.000} C_DIS
LIN {X 32.249,Y 30.327,Z 52.650,A 180.000,B 0.000,C 180.000} C_DIS
LIN {X 32.444,Y 30.194,Z 52.642,A 180.000,B 0.000,C 180.000} C_DIS
LIN {X 32.510,Y 30.152,Z 52.639,A 180.000,B 0.000,C 180.000} C_DIS
LIN {X 32.849,Y 29.951,Z 52.625,A 180.000,B 0.000,C 180.000} C_DIS
LIN {X 32.918,Y 29.913,Z 52.622,A 180.000,B 0.000,C 180.000} C_DIS
LIN {X 33.128,Y 29.806,Z 52.614,A 180.000,B 0.000,C 180.000} C_DIS
LIN {X 33.269,Y 29.734,Z 52.609,A 180.000,B 0.000,C 180.000} C_DIS
LIN {X 33.340,Y 29.701,Z 52.606,A 180.000,B 0.000,C 180.000} C_DIS
LIN {X 33.701,Y 29.544,Z 52.592,A 180.000,B 0.000,C 180.000} C_DIS
LIN {X 33.775,Y 29.515,Z 52.589,A 180.000,B 0.000,C 180.000} C_DIS
LIN {X 34.145,Y 29.382,Z 52.576,A 180.000,B 0.000,C 180.000} C_DIS
LIN {X 34.220,Y 29.357,Z 52.573,A 180.000,B 0.000,C 180.000} C_DIS
LIN {X 34.598,Y 29.248,Z 52.559,A 180.000,B 0.000,C 180.000} C_DIS
LIN {X 34.674,Y 29.228,Z 52.556,A 180.000,B 0.000,C 180.000} C_DIS
LIN {X 35.059,Y 29.142,Z 52.543,A 180.000,B 0.000,C 180.000} C_DIS
LIN {X 35.136,Y 29.128,Z 52.540,A 180.000,B 0.000,C 180.000} C_DIS
LIN {X 35.525,Y 29.066,Z 52.526,A 180.000,B 0.000,C 180.000} C_DIS
LIN {X 35.603,Y 29.056,Z 52.523,A 180.000,B 0.000,C 180.000} C_DIS
LIN {X 35.995,Y 29.019,Z 52.510,A 180.000,B 0.000,C 180.000} C_DIS
LIN {X 36.074,Y 29.015,Z 52.507,A 180.000,B 0.000,C 180.000} C_DIS
LIN {X 36.467,Y 29.002,Z 52.493,A 180.000,B 0.000,C 180.000} C_DIS
LIN {X 36.546,Y 29.003,Z 52.490,A 180.000,B 0.000,C 180.000} C_DIS
LIN {X 36.940,Y 29.015,Z 52.477,A 180.000,B 0.000,C 180.000} C_DIS
LIN {X 37.018,Y 29.021,Z 52.474,A 180.000,B 0.000,C 180.000} C_DIS
LIN {X 37.410,Y 29.058,Z 52.460,A 180.000,B 0.000,C 180.000} C_DIS
LIN {X 37.488,Y 29.068,Z 52.457,A 180.000,B 0.000,C 180.000} C_DIS
LIN {X 37.877,Y 29.130,Z 52.444,A 180.000,B 0.000,C 180.000} C_DIS
LIN {X 37.954,Y 29.145,Z 52.441,A 180.000,B 0.000,C 180.000} C_DIS
LIN {X 38.339,Y 29.231,Z 52.427,A 180.000,B 0.000,C 180.000} C_DIS
LIN {X 38.415,Y 29.251,Z 52.424,A 180.000,B 0.000,C 180.000} C_DIS
LIN {X 38.642,Y 29.317,Z 52.416,A 180.000,B 0.000,C 180.000} C_DIS
LIN {X 38.793,Y 29.361,Z 52.411,A 180.000,B 0.000,C 180.000} C_DIS
LIN {X 38.868,Y 29.386,Z 52.408,A 180.000,B 0.000,C 180.000} C_DIS
LIN {X 39.238,Y 29.520,Z 52.394,A 180.000,B 0.000,C 180.000} C_DIS
LIN {X 39.311,Y 29.550,Z 52.391,A 180.000,B 0.000,C 180.000} C_DIS
LIN {X 39.455,Y 29.612,Z 52.386,A 180.000,B 0.000,C 180.000} C_DIS
LIN {X 39.672,Y 29.706,Z 52.378,A 180.000,B 0.000,C 180.000} C_DIS
LIN {X 39.743,Y 29.741,Z 52.375,A 180.000,B 0.000,C 180.000} C_DIS
LIN {X 40.094,Y 29.919,Z 52.361,A 180.000,B 0.000,C 180.000} C_DIS
LIN {X 40.162,Y 29.958,Z 52.358,A 180.000,B 0.000,C 180.000} C_DIS
LIN {X 40.298,Y 30.038,Z 52.353,A 180.000,B 0.000,C 180.000} C_DIS
LIN {X 40.501,Y 30.159,Z 52.345,A 180.000,B 0.000,C 180.000} C_DIS
LIN {X 40.567,Y 30.202,Z 52.342,A 180.000,B 0.000,C 180.000} C_DIS
LIN {X 40.893,Y 30.423,Z 52.328,A 180.000,B 0.000,C 180.000} C_DIS
LIN {X 40.956,Y 30.471,Z 52.325,A 180.000,B 0.000,C 180.000} C_DIS
LIN {X 41.018,Y 30.519,Z 52.323,A 180.000,B 0.000,C 180.000} C_DIS
LIN {X 41.142,Y 30.615,Z 52.317,A 180.000,B 0.000,C 180.000} C_DIS
LIN {X 41.267,Y 30.712,Z 52.312,A 180.000,B 0.000,C 180.000} C_DIS
LIN {X 41.327,Y 30.763,Z 52.309,A 180.000,B 0.000,C 180.000} C_DIS
LIN {X 41.445,Y 30.867,Z 52.303,A 180.000,B 0.000,C 180.000} C_DIS
LIN {X 41.504,Y 30.920,Z 52.301,A 180.000,B 0.000,C 180.000} C_DIS
LIN {X 41.622,Y 31.024,Z 52.295,A 180.000,B 0.000,C 180.000} C_DIS
LIN {X 41.678,Y 31.079,Z 52.292,A 180.000,B 0.000,C 180.000} C_DIS
LIN {X 41.734,Y 31.134,Z 52.290,A 180.000,B 0.000,C 180.000} C_DIS
LIN {X 41.845,Y 31.246,Z 52.284,A 180.000,B 0.000,C 180.000} C_DIS
LIN {X 41.957,Y 31.357,Z 52.279,A 180.000,B 0.000,C 180.000} C_DIS
LIN {X 42.010,Y 31.416,Z 52.276,A 180.000,B 0.000,C 180.000} C_DIS
LIN {X 42.114,Y 31.534,Z 52.270,A 180.000,B 0.000,C 180.000} C_DIS
LIN {X 42.166,Y 31.593,Z 52.268,A 180.000,B 0.000,C 180.000} C_DIS
LIN {X 42.270,Y 31.711,Z 52.262,A 180.000,B 0.000,C 180.000} C_DIS
LIN {X 42.319,Y 31.773,Z 52.259,A 180.000,B 0.000,C 180.000} C_DIS
LIN {X 42.367,Y 31.835,Z 52.257,A 180.000,B 0.000,C 180.000} C_DIS
LIN {X 42.464,Y 31.960,Z 52.251,A 180.000,B 0.000,C 180.000} C_DIS
LIN {X 42.560,Y 32.084,Z 52.246,A 180.000,B 0.000,C 180.000} C_DIS
LIN {X 42.605,Y 32.149,Z 52.243,A 180.000,B 0.000,C 180.000} C_DIS
LIN {X 42.694,Y 32.279,Z 52.237,A 180.000,B 0.000,C 180.000} C_DIS
LIN {X 42.738,Y 32.344,Z 52.235,A 180.000,B 0.000,C 180.000} C_DIS
LIN {X 42.826,Y 32.474,Z 52.229,A 180.000,B 0.000,C 180.000} C_DIS
LIN {X 42.867,Y 32.542,Z 52.226,A 180.000,B 0.000,C 180.000} C_DIS
LIN {X 42.907,Y 32.610,Z 52.224,A 180.000,B 0.000,C 180.000} C_DIS
LIN {X 42.987,Y 32.745,Z 52.218,A 180.000,B 0.000,C 180.000} C_DIS
LIN {X 43.067,Y 32.881,Z 52.213,A 180.000,B 0.000,C 180.000} C_DIS
LIN {X 43.104,Y 32.951,Z 52.210,A 180.000,B 0.000,C 180.000} C_DIS
LIN {X 43.175,Y 33.091,Z 52.204,A 180.000,B 0.000,C 180.000} C_DIS
LIN {X 43.211,Y 33.161,Z 52.202,A 180.000,B 0.000,C 180.000} C_DIS
LIN {X 43.282,Y 33.302,Z 52.196,A 180.000,B 0.000,C 180.000} C_DIS
LIN {X 43.314,Y 33.374,Z 52.193,A 180.000,B 0.000,C 180.000} C_DIS
LIN {X 43.439,Y 33.663,Z 52.182,A 180.000,B 0.000,C 180.000} C_DIS
LIN {X 43.470,Y 33.735,Z 52.180,A 180.000,B 0.000,C 180.000} C_DIS
LIN {X 43.497,Y 33.809,Z 52.177,A 180.000,B 0.000,C 180.000} C_DIS
LIN {X 43.551,Y 33.957,Z 52.172,A 180.000,B 0.000,C 180.000} C_DIS
LIN {X 43.604,Y 34.106,Z 52.166,A 180.000,B 0.000,C 180.000} C_DIS
LIN {X 43.631,Y 34.180,Z 52.164,A 180.000,B 0.000,C 180.000} C_DIS
LIN {X 43.653,Y 34.255,Z 52.161,A 180.000,B 0.000,C 180.000} C_DIS
LIN {X 43.675,Y 34.331,Z 52.159,A 180.000,B 0.000,C 180.000} C_DIS
LIN {X 43.697,Y 34.407,Z 52.156,A 180.000,B 0.000,C 180.000} C_DIS
LIN {X 43.719,Y 34.482,Z 52.154,A 180.000,B 0.000,C 180.000} C_DIS
LIN {X 43.741,Y 34.558,Z 52.151,A 180.000,B 0.000,C 180.000} C_DIS
LIN {X 43.763,Y 34.633,Z 52.149,A 180.000,B 0.000,C 180.000} C_DIS
LIN {X 43.797,Y 34.787,Z 52.144,A 180.000,B 0.000,C 180.000} C_DIS
LIN {X 43.832,Y 34.941,Z 52.139,A 180.000,B 0.000,C 180.000} C_DIS
LIN {X 43.866,Y 35.095,Z 52.134,A 180.000,B 0.000,C 180.000} C_DIS
LIN {X 43.891,Y 35.250,Z 52.129,A 180.000,B 0.000,C 180.000} C_DIS
LIN {X 43.915,Y 35.406,Z 52.124,A 180.000,B 0.000,C 180.000} C_DIS
LIN {X 43.940,Y 35.561,Z 52.120,A 180.000,B 0.000,C 180.000} C_DIS
LIN {X 43.955,Y 35.718,Z 52.115,A 180.000,B 0.000,C 180.000} C_DIS
LIN {X 43.969,Y 35.875,Z 52.111,A 180.000,B 0.000,C 180.000} C_DIS
LIN {X 43.984,Y 36.032,Z 52.106,A 180.000,B 0.000,C 180.000} C_DIS
LIN {X 43.989,Y 36.189,Z 52.102,A 180.000,B 0.000,C 180.000} C_DIS
LIN {X 43.994,Y 36.347,Z 52.097,A 180.000,B 0.000,C 180.000} C_DIS
LIN {X 43.999,Y 36.504,Z 52.093,A 180.000,B 0.000,C 180.000} C_DIS
LIN {X 43.994,Y 36.662,Z 52.089,A 180.000,B 0.000,C 180.000} C_DIS
LIN {X 43.989,Y 36.819,Z 52.085,A 180.000,B 0.000,C 180.000} C_DIS
LIN {X 43.983,Y 36.976,Z 52.081,A 180.000,B 0.000,C 180.000} C_DIS
LIN {X 43.969,Y 37.133,Z 52.077,A 180.000,B 0.000,C 180.000} C_DIS
LIN {X 43.954,Y 37.290,Z 52.073,A 180.000,B 0.000,C 180.000} C_DIS
LIN {X 43.939,Y 37.447,Z 52.070,A 180.000,B 0.000,C 180.000} C_DIS
LIN {X 43.914,Y 37.602,Z 52.066,A 180.000,B 0.000,C 180.000} C_DIS
LIN {X 43.889,Y 37.758,Z 52.062,A 180.000,B 0.000,C 180.000} C_DIS
LIN {X 43.864,Y 37.914,Z 52.059,A 180.000,B 0.000,C 180.000} C_DIS
LIN {X 43.830,Y 38.067,Z 52.056,A 180.000,B 0.000,C 180.000} C_DIS
LIN {X 43.795,Y 38.221,Z 52.052,A 180.000,B 0.000,C 180.000} C_DIS
LIN {X 43.760,Y 38.375,Z 52.049,A 180.000,B 0.000,C 180.000} C_DIS
LIN {X 43.716,Y 38.526,Z 52.046,A 180.000,B 0.000,C 180.000} C_DIS
LIN {X 43.672,Y 38.677,Z 52.043,A 180.000,B 0.000,C 180.000} C_DIS
LIN {X 43.628,Y 38.828,Z 52.040,A 180.000,B 0.000,C 180.000} C_DIS
LIN {X 43.574,Y 38.976,Z 52.037,A 180.000,B 0.000,C 180.000} C_DIS
LIN {X 43.521,Y 39.124,Z 52.034,A 180.000,B 0.000,C 180.000} C_DIS
LIN {X 43.467,Y 39.272,Z 52.032,A 180.000,B 0.000,C 180.000} C_DIS
LIN {X 43.404,Y 39.417,Z 52.029,A 180.000,B 0.000,C 180.000} C_DIS
LIN {X 43.342,Y 39.562,Z 52.027,A 180.000,B 0.000,C 180.000} C_DIS
LIN {X 43.207,Y 39.846,Z 52.022,A 180.000,B 0.000,C 180.000} C_DIS
LIN {X 43.063,Y 40.126,Z 52.018,A 180.000,B 0.000,C 180.000} C_DIS
LIN {X 42.903,Y 40.397,Z 52.014,A 180.000,B 0.000,C 180.000} C_DIS
LIN {X 42.733,Y 40.663,Z 52.011,A 180.000,B 0.000,C 180.000} C_DIS
LIN {X 42.555,Y 40.923,Z 52.008,A 180.000,B 0.000,C 180.000} C_DIS
LIN {X 42.362,Y 41.171,Z 52.005,A 180.000,B 0.000,C 180.000} C_DIS
LIN {X 42.160,Y 41.413,Z 52.003,A 180.000,B 0.000,C 180.000} C_DIS
LIN {X 41.951,Y 41.649,Z 52.002,A 180.000,B 0.000,C 180.000} C_DIS
LIN {X 41.728,Y 41.871,Z 52.001,A 180.000,B 0.000,C 180.000} C_DIS
LIN {X 41.498,Y 42.086,Z 52.000,A 180.000,B 0.000,C 180.000} C_DIS
LIN {X 41.323,Y 42.240,Z 52.000,A 180.000,B 0.000,C 180.000} C_DIS
; Cutting Move Starts
LIN {X 41.299,Y 42.261,Z 52.000,A 180.000,B 0.000,C 180.000} C_DIS
LIN {X 41.159,Y 42.372,Z 52.000,A 180.000,B 0.000,C 180.000} C_DIS
LIN {X 40.928,Y 42.550,Z 52.000,A 180.000,B 0.000,C 180.000} C_DIS
LIN {X 40.763,Y 42.665,Z 52.000,A 180.000,B 0.000,C 180.000} C_DIS
LIN {X 40.584,Y 42.787,Z 52.000,A 180.000,B 0.000,C 180.000} C_DIS
LIN {X 40.405,Y 42.898,Z 52.000,A 180.000,B 0.000,C 180.000} C_DIS
LIN {X 40.226,Y 43.004,Z 52.000,A 180.000,B 0.000,C 180.000} C_DIS
LIN {X 40.082,Y 43.087,Z 52.000,A 180.000,B 0.000,C 180.000} C_DIS
LIN {X 39.731,Y 43.266,Z 52.000,A 180.000,B 0.000,C 180.000} C_DIS
LIN {X 39.690,Y 43.286,Z 52.000,A 180.000,B 0.000,C 180.000} C_DIS
LIN {X 39.325,Y 43.444,Z 52.000,A 180.000,B 0.000,C 180.000} C_DIS
LIN {X 39.154,Y 43.511,Z 52.000,A 180.000,B 0.000,C 180.000} C_DIS
LIN {X 38.841,Y 43.623,Z 52.000,A 180.000,B 0.000,C 180.000} C_DIS
LIN {X 38.796,Y 43.638,Z 52.000,A 180.000,B 0.000,C 180.000} C_DIS
LIN {X 38.439,Y 43.742,Z 52.000,A 180.000,B 0.000,C 180.000} C_DIS
LIN {X 38.260,Y 43.787,Z 52.000,A 180.000,B 0.000,C 180.000} C_DIS
LIN {X 38.081,Y 43.827,Z 52.000,A 180.000,B 0.000,C 180.000} C_DIS
LIN {X 37.902,Y 43.866,Z 52.000,A 180.000,B 0.000,C 180.000} C_DIS
LIN {X 37.545,Y 43.923,Z 52.000,A 180.000,B 0.000,C 180.000} C_DIS
LIN {X 37.366,Y 43.947,Z 52.000,A 180.000,B 0.000,C 180.000} C_DIS
LIN {X 37.006,Y 43.981,Z 52.000,A 180.000,B 0.000,C 180.000} C_DIS
LIN {X 36.830,Y 43.988,Z 52.000,A 180.000,B 0.000,C 180.000} C_DIS
LIN {X 36.651,Y 43.994,Z 52.000,A 180.000,B 0.000,C 180.000} C_DIS
LIN {X 36.472,Y 43.998,Z 52.000,A 180.000,B 0.000,C 180.000} C_DIS
LIN {X 36.115,Y 43.987,Z 52.000,A 180.000,B 0.000,C 180.000} C_DIS
LIN {X 35.994,Y 43.981,Z 52.000,A 180.000,B 0.000,C 180.000} C_DIS
LIN {X 35.578,Y 43.941,Z 52.000,A 180.000,B 0.000,C 180.000} C_DIS
LIN {X 35.400,Y 43.914,Z 52.000,A 180.000,B 0.000,C 180.000} C_DIS
LIN {X 35.221,Y 43.886,Z 52.000,A 180.000,B 0.000,C 180.000} C_DIS
LIN {X 35.042,Y 43.854,Z 52.000,A 180.000,B 0.000,C 180.000} C_DIS
LIN {X 34.685,Y 43.774,Z 52.000,A 180.000,B 0.000,C 180.000} C_DIS
LIN {X 34.506,Y 43.726,Z 52.000,A 180.000,B 0.000,C 180.000} C_DIS
LIN {X 34.327,Y 43.674,Z 52.000,A 180.000,B 0.000,C 180.000} C_DIS
LIN {X 34.159,Y 43.623,Z 52.000,A 180.000,B 0.000,C 180.000} C_DIS
LIN {X 33.791,Y 43.491,Z 52.000,A 180.000,B 0.000,C 180.000} C_DIS
